// SIMATIC S7-200 project (STEP 7-Micro/WIN), CPU 226 CN REL 02.01

SYMBOL_TABLE INPUT
HMI_ES           I0.0     // HMI急停
WORK_START       I0.1     // 开始工作
BP_ES_RESET      I0.2     // 急停复位
BP_DOOR_RESET    I0.3     // 安全门复位
BP_MANUAL        I0.4     // 手动
BP_AUTO          I0.5     // 自动
BP_START         I0.6     // 启动
ES_OK            I0.7
BP_ES            I1.0     // 操作盒急停
BP_DOOR_PRESET   I1.1     // 安全门预约
AS_OK            I1.2
BP_DOOR_RESET1   I1.3     // 门复位
CS1              I1.4
CS2              I1.5
CS3              I1.6
CS4              I1.7
A伺服就绪            I2.0
A定位结束            I2.1
DSL1             I2.2
DSL2             I2.3
B伺服就绪            I2.4
B定位结束            I2.5
DSR1             I2.6
DSR2             I2.7
BV1_1A           I3.0
BV1_1B           I3.1
BV1_2A           I3.2
BV1_2B           I3.3
BS1              I3.4
BS2              I3.5
B行程保护            I3.6
A请求夹紧            I3.7     // A-R2夹紧请求
BV2_1A           I4.0
BV2_1B           I4.1
BV2_2A           I4.2
BV2_2B           I4.3
BV3_1A           I4.4
BV3_1B           I4.5
BS3              I4.6
B请求夹紧            I4.7     // B-R2夹紧请求
R1_AUTO          I5.0
R1_CYCLE_NO      I5.1
R1_IN_JOB1       I5.2
R1_IN_JOB2       I5.3
R1_HOME          I5.4
R1_ES_OK         I5.5
R1_IN_UNLOAD     I5.6     // 机器人开始抓件
R1_FINISH3       I5.7     // 机器人抓件完成
R1_FINISH1       I6.0     // 机器人放件完成
R1_FINISH2       I6.1     // 机器人取件完成
IN_R1_POS1       I6.2     // 伺服位置返回信号－－产品
IN_R1_POS2       I6.3     // 伺服位置返回信号
IN_R1_POS3       I6.4     // 伺服位置返回信号
IN_R1_POS4       I6.5     // 伺服位置返回信号
IN_R1_PIC1       I6.6     // 机器人返回组信号－－偏差
IN_R1_PIC2       I6.7     // 机器人返回组信号
R2_AUTO          I7.0     // 机器人自动
R2_CYCLE_NO      I7.1     // 机器人上电
R2_IN_JOB1       I7.2
R2_IN_JOB2       I7.3
R2_HOME          I7.4
R2_ES_OK         I7.5     // 机器人急停正常
R2_工位1           I7.6     // A－变位机位置
R2_工位2           I7.7     // B－变位机位置
R2_FINISH1       I8.0     // 机器人2抓件完成
R2_FINISH2       I8.1     // 机器人2焊接完成
IN_R2_POS1       I8.2     // 伺服位置返回信号－－产品
IN_R2_POS2       I8.3     // 伺服位置返回信号
IN_R2_POS3       I8.4     // 伺服位置返回信号
IN_R2_POS4       I8.5     // 伺服位置返回信号
IN_R2_PIC1       I8.6     // 机器人返回组信号－－偏差
IN_R2_PIC2       I8.7     // 机器人返回组信号
AV1_1A           I9.0
AV1_1B           I9.1
AV1_2A           I9.2
AV1_2B           I9.3
AS1              I9.4
AS2              I9.5
A行程保护            I9.6
CV2_A            I9.7     // 横梁传送检测汽缸夹紧信号
AV2_1A           I10.0
AV2_1B           I10.1
AV2_2A           I10.2
AV2_2B           I10.3
AV3_1A           I10.4
AV3_1B           I10.5
AS3              I10.6
END_SYMBOL_TABLE

SYMBOL_TABLE OUTPUT
WORK_H           Q0.0     // 工作指示
ES_H             Q0.1     // 急停复位指示
DOOR_H           Q0.2     // 安全门复位指示
START_H          Q0.3     // 自动启动指示
GN_H             Q0.5     // 绿灯
YE_H             Q0.6     // 黄灯
RD_H             Q0.7     // 红灯
CHECK_DUMMY      Q1.0     // 工件检测虚拟打开
DOOR_OUT         Q1.1     // 安全门
RESET_ES_OUT     Q1.2     // 急停复位输出
RESET_DOOR_OUT   Q1.3
R1_PRO_START     Q4.0     // 给机器人程序开始
RI_CYCLE_START   Q4.1     // 给机器人系统开始
R1_CYCLE_STOP    Q4.2     // 给机器人系统停止
R1_RESET_ES      Q4.3     // 复位机器人急停
R1_JOB1_VAILD    Q4.4     // 开始放件工作的号
R1_JOB2_VAILD    Q4.5     // 开始取件工作的号
R1_STAT1_OK      Q4.6     // 上夹具准备就绪
R1_STAT2_OK      Q4.7     // 下夹具准备就绪
R1_UNLOAD_OK     Q5.0     // 机器人抓件准备就绪
R1_JOB3_VALD     Q5.1     // 启动机器人抓件
R1_POS1          Q5.2     // 伺服位置组信号－－产品
R1_POS2          Q5.3     // 伺服位置组信号
R1_POS3          Q5.4     // 伺服位置组信号
R1_POS4          Q5.5     // 伺服位置组信号
R1_PIC1          Q5.6     // 工件组信号－－偏差
R1_PIC2          Q5.7     // 工件组信号
R2_PRO_START     Q6.0     // 给机器人程序开始
R2_CYCLE_START   Q6.1     // 给机器人系统开始
R2_CYCLE_STOP    Q6.2     // 给机器人系统停止
R2_RESET_ES      Q6.3     // 复位机器人急停
R2_JOB1_VAILD    Q6.4     // 开始放件程序
R2_JOB2_VAILD    Q6.5     // 开始焊接程序
R2_STAT1_OK      Q6.6     // 上夹具准备就绪,可以装件
R2_STAT2_OK      Q6.7     // 下夹具准备就绪,可以装件
R2_A_小件夹紧        Q7.0     // 放小件夹紧A
R2_B_小件夹紧        Q7.1     // 放小件夹紧B
R2_POS1          Q7.2     // 伺服位置组信号－－产品
R2_POS2          Q7.3     // 伺服位置组信号
R2_POS3          Q7.4     // 伺服位置组信号
R2_POS4          Q7.5     // 伺服位置组信号
R2_PIC1          Q7.6     // 工件组信号－－偏差
R2_PIC2          Q7.7     // 工件组信号
AV1_A            Q8.0
AV1_B            Q8.1
AV2_A            Q8.4
AV2_B            Q8.5
AV3_A            Q8.6
AV3_B            Q8.7
BV1_A            Q10.0
BV1_B            Q10.1
BV2_A            Q10.4
BV2_B            Q10.5
BV3_A            Q10.6
BV3_B            Q10.7
A_SRV_ON         Q11.0    // 伺服1使能
A_CLR            Q11.1    // 伺服1报警清除
B_SRV_ON         Q11.2    // 伺服2使能
B_CLR            Q11.3    // 伺服2报警清除
END_SYMBOL_TABLE

SYMBOL_TABLE SERVICE_A
A_MOD_EN         V540.0
A_MAN_RUN        V540.1
A_JOG_P          V540.2
A_JOG_N          V540.3
A_MAN_DIR        V540.4
A_MAN_DONE       V540.5
A_GOTO_START     V540.6
A_GOTO_ABORT     V540.7
A_GOTO_DONE      V541.0
A_RUN_START1     V541.1
A_RUN_ABORT1     V541.2
A_RUN_DONE1      V541.3
A_RUN_START2     V541.4
A_RUN_ABORT2     V541.5
A_RUN_DONE2      V541.6
A_RUN_START3     V541.7
A_RUN_ABORT3     V542.0
A_RUN_DONE3      V542.1
A_RUN_START4     V542.2
A_RUN_ABORT4     V542.3
A_RUN_DONE4      V542.4
A_RUN_START5     V542.5
A_RUN_ABORT5     V542.6
A_RUN_DONE5      V542.7
A_RUN_START6     V543.0
A_RUN_ABORT6     V543.1
A_RUN_DONE6      V543.2
A_RUN_START7     V543.3
A_RUN_ABORT7     V543.4
A_RUN_DONE7      V543.5
A_RUN_START8     V543.6
A_RUN_ABORT8     V543.7
A_RUN_DONE8      V544.0
A_RSEEK_START    V545.0
A_RSEEK_DONE     V545.1
A_DONE           V550.0
A_C_DIR          V550.1
A_ERROR          VB551
A_POS            VD552
A_SPEED          VD556
A_GOTO_ERR       VB560
A_GOTO_C_POS     VD562
A_GOTO_C_SPEED   VD566
A_RUN_ERR        VB570
A_RUN_C_PROF     VB571
A_RUN_C_STEP     VB572
A_RUN_C_POS      VD574
A_RUN_C_SPEED    VD578
A_MAN_SPEED      VD586
A_GOTO_POS       VD590
A_GOTO_SPEED     VD594
A_GOTO_MODE      VB598
A补偿启动            V820.0
A补偿位置            VD822
A补偿速度            VD826
A绝对位置            VD832
A绝对速度            VD836
END_SYMBOL_TABLE

SYMBOL_TABLE UP_A
AV1夹紧的命令         V500.0
AV1夹紧的条件         V500.1
AV1夹紧            V500.2
HMI_AV1夹紧        V500.3
AV1全部夹紧          V500.7
AV1放松的命令         V501.0
AV1放松的条件         V501.1
AV1放松            V501.2
HMI_AV1放松        V501.3
AV1全部放松          V501.7
AV2夹紧的命令         V502.0
AV2夹紧的条件         V502.1
AV2夹紧            V502.2
HMI_AV2夹紧        V502.3
AV2全部夹紧          V502.7
AV2放松的命令         V503.0
AV2放松的条件         V503.1
AV2放松            V503.2
HMI_AV2放松        V503.3
AV2全部放松          V503.7
AV3夹紧的命令         V504.0
AV3夹紧的条件         V504.1
AV3夹紧            V504.2
HMI_AV3夹紧        V504.3
HMI_AV3_MAN_断电   V504.4
AV3全部夹紧          V504.7
AV3放松的命令         V505.0
AV3放松的条件         V505.1
AV3放松            V505.2
HMI_AV3放松        V505.3
AV3全部放松          V505.7
AV大件偏短           V508.0
AV大件偏长           V508.1
AV焊接偏短           V508.2
AV焊接偏长           V508.3
AV取件偏短           V508.4
AV取件偏长           V508.5
AV夹紧             V510.0
AV全部夹紧           V510.1
AV全部放松           V510.2
AV预约             V510.3
AV有小件            V510.4
AV有大件            V510.5
AV有件             V510.6
AV未装件            V510.7
AV放小件准备就绪        V511.0
AV放小件            V511.1
AV请求夹紧           V511.2
AV放小件完成          V511.3
AV放大件准备就绪        V511.4
AV放大件            V511.5
AV放大件完成          V511.6
AV焊接准备就绪         V511.7
AV焊接             V512.0
AV焊接完成           V512.1
AV还原准备           V512.2
AV夹具还原           V512.3
AV取件准备就绪         V512.4
AV取件             V512.5
AV取件完成           V512.6
A_JOB_NUM        VW514
END_SYMBOL_TABLE

SYMBOL_TABLE DOWM_B
BV1夹紧的命令         V600.0
BV1夹紧的条件         V600.1
BV1夹紧            V600.2
HMI_BV1夹紧        V600.3
BV1全部夹紧          V600.7
BV1放松的命令         V601.0
BV1放松的条件         V601.1
BV1放松            V601.2
HMI_BV1放松        V601.3
BV1全部放松          V601.7
BV2夹紧的命令         V602.0
BV2夹紧的条件         V602.1
BV2夹紧            V602.2
HMI_BV2夹紧        V602.3
BV2全部夹紧          V602.7
BV2放松的命令         V603.0
BV2放松的条件         V603.1
BV2放松            V603.2
HMI_BV2放松        V603.3
BV2全部放松          V603.7
BV3夹紧的命令         V604.0
BV3夹紧的条件         V604.1
BV3夹紧            V604.2
HMI_BV3夹紧        V604.3
HMI_BV3_MAN_断电   V604.4
BV3全部夹紧          V604.7
BV3放松的命令         V605.0
BV3放松的条件         V605.1
BV3放松            V605.2
HMI_BV3放松        V605.3
BV3全部放松          V605.7
BV大件偏短           V608.0
BV大件偏长           V608.1
BV焊接偏短           V608.2
BV焊接偏长           V608.3
BV取件偏短           V608.4
BV取件偏长           V608.5
BV夹紧             V610.0
BV全部夹紧           V610.1
BV全部放松           V610.2
BV预约             V610.3
BV有小件            V610.4
BV有大件            V610.5
BV有件             V610.6
BV未装件            V610.7
BV放小件准备就绪        V611.0
BV放小件            V611.1
BV请求夹紧           V611.2
BV放小件完成          V611.3
BV放大件准备就绪        V611.4
BV放大件            V611.5
BV放大件完成          V611.6
BV焊接准备就绪         V611.7
BV焊接             V612.0
BV焊接完成           V612.1
BV还原准备           V612.2
BV夹具还原           V612.3
BV取件准备就绪         V612.4
BV取件             V612.5
BV取件完成           V612.6
B_JOB_NUM        VW614
END_SYMBOL_TABLE

SYMBOL_TABLE SERVICE_B
B_MOD_EN         V640.0
B_MAN_RUN        V640.1
B_JOG_P          V640.2
B_JOG_N          V640.3
B_MAN_DIR        V640.4
B_MAN_DONE       V640.5
B_GOTO_START     V640.6
B_GOTO_ABORT     V640.7
B_GOTO_DONE      V641.0
B_RUN_START1     V641.1
B_RUN_ABORT1     V641.2
B_RUN_DONE1      V641.3
B_RUN_START2     V641.4
B_RUN_ABORT2     V641.5
B_RUN_DONE2      V641.6
B_RUN_START3     V641.7
B_RUN_ABORT3     V642.0
B_RUN_DONE3      V642.1
B_RUN_START4     V642.2
B_RUN_ABORT4     V642.3
B_RUN_DONE4      V642.4
B_RUN_START5     V642.5
B_RUN_ABORT5     V642.6
B_RUN_DONE5      V642.7
B_RUN_START6     V643.0
B_RUN_ABORT6     V643.1
B_RUN_DONE6      V643.2
B_RUN_START7     V643.3
B_RUN_ABORT7     V643.4
B_RUN_DONE7      V643.5
B_RUN_START8     V643.6
B_RUN_ABORT8     V643.7
B_RUN_DONE8      V644.0
B_RSEEK_START    V645.0
B_RSEEK_DONE     V645.1
B_DONE           V650.0
B_C_DIR          V650.1
B_ERROR          VB651
B_POS            VD652
B_SPEED          VD656
B_GOTO_ERR       VB660
B_GOTO_C_POS     VD662
B_GOTO_C_SPEED   VD666
B_RUN_ERR        VB670
B_RUN_C_PROF     VB671
B_RUN_C_STEP     VB672
B_RUN_C_POS      VD674
B_RUN_C_SPEED    VD678
B_MAN_SPEED      VD686
B_GOTO_POS       VD690
B_GOTO_SPEED     VD694
B_GOTO_MODE      VB698
B补偿启动            V920.0
B补偿位置            VD922
B补偿速度            VD926
B绝对位置            VD932
B绝对速度            VD936
END_SYMBOL_TABLE

SYMBOL_TABLE INTERFACE
BV允许抓大件          M4.1
AV允许抓大件          M4.0
开始工作辅助           M0.1
开始工作             M0.0
HMI_RESET_ALARM  M1.0
HMI_LAMP_TEST    M1.1
HMI_RUN_FREE     M1.2
HMI_PAUSE        M1.3
HMI_ST1_PASS     M1.4
HMI_ST2_PASS     M1.5
HMI_INIT         M1.6     // 初始化－HMI
INIT             M1.7
INIT1_FINISH     M2.0
INIT2_FINISH     M2.1
INIT_FINISH      M2.2
PAUSE            M2.3
ST1_PASS         M2.4
ST1_PASS1        M2.5
ST2_PASS         M2.6
ST2_PASS1        M2.7
ST1_WORKING      M3.0
ST2_WORKING      M3.1
HMI_FINISH       M3.2
FINISH           M3.3
PRE_FINISH       M3.4
FINISHED         M3.5
AV_HOME          M3.6
BV_HOME          M3.7
HMI_A_SEV_ON     M5.0
HMI_A_SEV_OFF    M5.1
HMI_A_PIC        M5.2
HMI_B_SEV_ON     M6.0
HMI_B_SEV_OFF    M6.1
HMI_B_PIC        M6.2
绝对画面             M7.0
相对画面             M7.1
HMI_SEV_AB_ON    M8.0
HMI_SEV_AB_HOME  M8.1
NOAUTO           M10.0
AUTO             M10.1
ATUOSTART        M10.2
CONTROL_NO       M10.3
A1合格组信号1         M11.0
A1合格组信号2         M11.1
A2合格组信号1         M11.2
A2合格组信号2         M11.3
B1合格组信号1         M11.4
B1合格组信号2         M11.5
B2合格组信号1         M11.6
B2合格组信号2         M11.7
产品组信号1           M12.0
产品组信号2           M12.1
产品组信号3           M12.2
产品组信号4           M12.3
A工件合格            M14.0
A工件不合格           M14.1
A检测合格            M14.2
B工件合格            M14.4
B工件不合格           M14.5
B检测合格            M14.6
R1_IN_SAFE       M15.0
R1_START         M15.1
R1_JOB_READY     M15.4
R1_POS_OK        M15.5
R1_PIC_OK        M15.6
R1_抓件中           M16.0
R1_抓件完成          M16.1
R2_IN_SAFE       M17.0
R2_START         M17.1
R2_JOB_READY     M17.4
R2_POS_OK        M17.5
R2_PIC_OK        M17.6
A_HOME_POS       M20.0
B_HOME_POS       M22.0
R_IN_SAFE        M23.0
A_CRE_ACT        M30.0
B_CRE_ACT        M30.1
R1_CRE_ACT       M30.2
R2_CRE_ACT       M30.3
SERV_A_ACT       M30.4
SERV_B_ACT       M30.5
DUMMY            M31.0
虚拟               M31.2
虚拟reset          M31.3
PULSE_1          M31.4
HMI_产品选择1        V420.0
HMI_产品选择2        V420.1
HMI_产品选择3        V420.2
HMI_产品选择4        V420.3
HMI_产品选择5        V420.4
HMI_产品选择6        V420.5
HMI_产品选择7        V420.6
HMI_产品选择8        V420.7
HMI_产品选择9        V421.0
HMI_产品选择10       V421.1
HMI_产品选择11       V421.2
HMI_产品选择12       V421.3
HMI_产品选择13       V421.4
HMI_产品选择14       V421.5
HMI_产品选择15       V421.6
HMI_产品选择16       V421.7
产品选择1            V450.0
产品选择2            V450.1
产品选择3            V450.2
产品选择4            V450.3
产品选择5            V450.4
产品选择6            V450.5
产品选择7            V450.6
产品选择8            V450.7
产品选择9            V451.0
产品选择10           V451.1
产品选择11           V451.2
产品选择12           V451.3
产品选择13           V451.4
产品选择14           V451.5
产品选择15           V451.6
产品选择16           V451.7
A产品1             V460.0
A产品2             V460.1
A产品3             V460.2
A产品4             V460.3
A产品5             V460.4
A产品6             V460.5
A产品7             V460.6
A产品8             V460.7
A产品9             V461.0
A产品10            V461.1
A产品11            V461.2
A产品12            V461.3
A产品13            V461.4
A产品14            V461.5
A产品15            V461.6
A产品16            V461.7
B产品1             V462.0
B产品2             V462.1
B产品3             V462.2
B产品4             V462.3
B产品5             V462.4
B产品6             V462.5
B产品7             V462.6
B产品8             V462.7
B产品9             V463.0
B产品10            V463.1
B产品11            V463.2
B产品12            V463.3
B产品13            V463.4
B产品14            V463.5
B产品15            V463.6
B产品16            V463.7
P_放大件            V464.0
P_放小件            V464.1
放大件              V464.2
放小件              V464.3
放件确认             V465.0
放件取消             V465.1
产品选择显示           VB480
产品提示             VB470
选择产品1            V490.0
选择产品2            V490.1
选择产品3            V490.2
选择产品4            V490.3
选择产品5            V490.4
选择产品6            V490.5
选择产品7            V490.6
选择产品8            V490.7
选择产品9            V491.0
选择产品10           V491.1
选择产品11           V491.2
选择产品12           V491.3
选择产品13           V491.4
选择产品14           V491.5
选择产品15           V491.6
选择产品16           V491.7
传送检测气缸信号上        V530.0
检测CS1            V530.1
检测CS2            V530.2
检测CS3            V530.3
END_SYMBOL_TABLE

SYMBOL_TABLE MSSG
AV1_1A_MESS      V400.0
AV1_2A_MESS      V400.1
AV1_3A_MESS      V400.2
AV1_4A_MESS      V400.3
AV1_1B_MESS      V400.4
AV1_2B_MESS      V400.5
AV1_3B_MESS      V400.6
AV1_4B_MESS      V400.7
AV2_1A_MESS      V401.0
AV2_2A_MESS      V401.1
AV2_3A_MESS      V401.2
AV2_4A_MESS      V401.3
AV2_1B_MESS      V401.4
AV2_2B_MESS      V401.5
AV2_3B_MESS      V401.6
AV2_4B_MESS      V401.7
AV3_1A_MESS      V402.0
AV3_2A_MESS      V402.1
AV3_3A_MESS      V402.2
AV3_4A_MESS      V402.3
AV3_1B_MESS      V402.4
AV3_2B_MESS      V402.5
AV3_3B_MESS      V402.6
AV3_4B_MESS      V402.7
AV4_1A_MESS      V403.0
AV4_2A_MESS      V403.1
AV4_3A_MESS      V403.2
AV4_4A_MESS      V403.3
AV4_1B_MESS      V403.4
AV4_2B_MESS      V403.5
AV4_3B_MESS      V403.6
AV4_4B_MESS      V403.7
BV1_1A_MESS      V404.0
BV1_2A_MESS      V404.1
BV1_3A_MESS      V404.2
BV1_4A_MESS      V404.3
BV1_1B_MESS      V404.4
BV1_2B_MESS      V404.5
BV1_3B_MESS      V404.6
BV1_4B_MESS      V404.7
BV2_1A_MESS      V405.0
BV2_2A_MESS      V405.1
BV2_3A_MESS      V405.2
BV2_4A_MESS      V405.3
BV2_1B_MESS      V405.4
BV2_2B_MESS      V405.5
BV2_3B_MESS      V405.6
BV2_4B_MESS      V405.7
BV3_1A_MESS      V406.0
BV3_2A_MESS      V406.1
BV3_3A_MESS      V406.2
BV3_4A_MESS      V406.3
BV3_1B_MESS      V406.4
BV3_2B_MESS      V406.5
BV3_3B_MESS      V406.6
BV3_4B_MESS      V406.7
BV4_1A_MESS      V407.0
BV4_2A_MESS      V407.1
BV4_3A_MESS      V407.2
BV4_4A_MESS      V407.3
BV4_1B_MESS      V407.4
BV4_2B_MESS      V407.5
BV4_3B_MESS      V407.6
BV4_4B_MESS      V407.7
MESS65           V408.0   // 警报   AS1无感应
MESS66           V408.1   // 警报   AS1有感应
MESS67           V408.2   // AS2无感应
MESS68           V408.3   // AS2有感应
MESS69           V408.4   // AS3无感应
MESS70           V408.5   // AS3有感应
MESS71           V408.6   // AS4无感应
MESS72           V408.7   // AS4有感应
MESS73           V409.0   // BS1无感应警报
MESS74           V409.1   // BS1有感应警报
MESS75           V409.2   // BS2无感应
MESS76           V409.3   // BS2有感应
MESS77           V409.4   // BS3无感应
MESS78           V409.5   // BS3有感应
MESS79           V409.6   // BS4无感应
MESS80           V409.7   // BS4有感应
MESS81           V410.0   // CS1无感应警报
MESS82           V410.1   // CS1有感应警报
MESS83           V410.2   // CS2无感应
MESS84           V410.3   // CS2有感应
MESS85           V410.4   // CS3无感应
MESS86           V410.5   // CS3有感应
MESS87           V410.6   // CS4无感应
MESS88           V410.7   // CS4有感应
MESS89           V411.0   // DSL1无感应警报
MESS90           V411.1   // DSL1有感应警报
MESS91           V411.2   // DSL2无感应
MESS92           V411.3   // DSL2有感应
MESS93           V411.4   // DSR1无感应
MESS94           V411.5   // DSR1有感应
MESS95           V411.6   // DSR2无感应
MESS96           V411.7   // DSR2有感应
MESS97           V412.0
MESS98           V412.1
MESS99           V412.2
MESS100          V412.3
MESS101          V412.4
MESS102          V412.5
MESS103          V412.6
MESS104          V412.7
MESS105          V413.0
MESS106          V413.1
MESS107          V413.2
MESS108          V413.3
MESS109          V413.4
MESS110          V413.5
MESS111          V413.6
MESS112          V413.7
MESS113          V414.0   // A伺服电机未查找原点
MESS114          V414.1   // A伺服器未准备就绪
MESS115          V414.2   // A伺服器未上电
MESS116          V414.3   // B伺服电机未查找原点
MESS117          V414.4   // B伺服器未准备就绪
MESS118          V414.5   // B伺服器未上电
MESS119          V414.6   // 机器人1不在原点
MESS120          V414.7   // 机器人2不在原点
MESS121          V415.0   // 机器人1不在自动
MESS122          V415.1   // 机器人2不在自动
MESS123          V415.2   // 机器人1系统未运行
MESS124          V415.3   // 机器人2系统未运行
MESS125          V415.4   // 机器人2不在工位1
MESS126          V415.5   // 机器人2不在工位2
MESS127          V415.6   // A夹具上有工件
MESS128          V415.7   // B夹具上有工件
MESS129          V416.0   // 机器人1急停
MESS130          V416.1   // 机器人2急停
MESS131          V416.2   // 系统急停
MESS132          V416.3   // HMI操作箱急停
MESS133          V416.4   // 安全门操作盒急停
MESS134          V416.5   // 急停按钮未复位
MESS135          V416.6   // 安全打开状态
MESS136          V416.7   // 安全门需要复位
MESS137          V417.0   // 启动条件未满足
MESS138          V417.1
MESS139          V417.2
MESS140          V417.3
MESS141          V417.4
MESS142          V417.5
MESS143          V417.6
MESS144          V417.7
MESS145          V418.0   // 系统空运行测试
MESS146          V418.1   // 夹具1被屏蔽
MESS147          V418.2   // 夹具2被屏蔽
MESS148          V418.3   // 系统暂停运行
MESS149          V418.4   // 系统运行结束
MESS150          V418.5
MESS151          V418.6
MESS152          V418.7
MESS153          V419.0
MESS154          V419.1
MESS155          V419.2
MESS156          V419.3
MESS157          V419.4
MESS158          V419.5
MESS159          V419.6
MESS160          V419.7
AV1_A_CAT        V422.0
AV1_B_CAT        V422.1
AV2_A_CAT        V422.2
AV2_B_CAT        V422.3
AV3_A_CAT        V422.4
AV3_B_CAT        V422.5
AV4_A_CAT        V422.6
AV4_B_CAT        V422.7
BV1_A_CAT        V423.0
BV1_B_CAT        V423.1
BV2_A_CAT        V423.2
BV2_B_CAT        V423.3
BV3_A_CAT        V423.4
BV3_B_CAT        V423.5
BV4_A_CAT        V423.6
BV4_B_CAT        V423.7
AV1_A_RES        V426.0
AV1_B_RES        V426.1
AV2_A_RES        V426.2
AV2_B_RES        V426.3
AV3_A_RES        V426.4
AV3_B_RES        V426.5
AV4_A_RES        V426.6
AV4_B_RES        V426.7
BV1_A_RES        V427.0
BV1_B_RES        V427.1
BV2_A_RES        V427.2
BV2_B_RES        V427.3
BV3_A_RES        V427.4
BV3_B_RES        V427.5
BV4_A_RES        V427.6
BV4_B_RES        V427.7
画面号              VW752
END_SYMBOL_TABLE

ORGANIZATION_BLOCK 主程序:OB1
TITLE=PLC程序用于控制一个自动化生产线，通过两个EM253模块控制松下伺服电机A和B，定位工件长度，并协调搬运机器人和焊接机器人完成生产任务。设备包括松下伺服电机A和B、搬运机器人、焊接机器人、传感器、按钮和指示灯。
// HMI初始化信号由HMI界面触发。系统通过HMI初始化信号启动操作界面，并需确保急停按钮状态未被按下，以保证系统安全运行。操作员可通过手动模式开关或自动模式开关选择运行模式。在手动模式下，操作员可以直接控制夹具的夹紧和放松以及伺服电机的开关。而在自动模式下，启动按钮触发整个生产流程，伺服电机A驱动工位1的工件定位，伺服电机B驱动工位2的工件定位，且需在急停按钮状态正常时激活，以避免设备失控。
// 生产过程中，系统实时监控工位1和工位2的工作状态，并根据A夹具和B夹具的未装件状态判断夹具是否就绪。机器人1开始抓取信号由机器人控制器发出。搬运机器人（机器人1）根据夹具状态执行工件搬运任务，例如，当机器人1开始抓取信号置位时，系统需确认A夹具状态达到指定位置，确保工件正确定位后抓取。随后，焊接机器人（机器人2）在夹具完成夹紧后进行焊接。A夹具工件检测结果用于记录工件长度检测的数据。工件长度检测是关键环节，当传送检测气缸信号为真且工位1和工位2的工作状态均为假时，系统记录A夹具和B夹具的工件检测结果，以确保数据准确。
// 若夹具动作异常，例如伺服电机A的夹紧输出触发失败，A夹具错误计数器会递增以记录异常次数。为了避免误报警影响生产稳定性，系统会在生产周期结束时清零A夹具错误计数器。整个流程结束后，生产周期结束标志置位，系统进入待机状态，等待下一次启动。急停按钮状态若被按下，所有操作立即停止，确保车间人员和设备的安全。
BEGIN
Network 1
LD     SM0.0
CALL   INTERFACE:SBR0
Network 2
LD     SM0.0
CALL   AV1:SBR1
Network 3
LD     SM0.0
CALL   AV2:SBR2
Network 4
LD     SM0.0
CALL   AV3:SBR3
Network 5
LD     SM0.0
CALL   BV1:SBR4
Network 6
LD     SM0.0
CALL   BV2:SBR5
Network 7
LD     SM0.0
CALL   BV3:SBR6
Network 8
LD     A_SRV_ON:Q11.0
CALL   SERVICE_A:SBR7
Network 9
LD     B_SRV_ON:Q11.2
CALL   SERVICEE_B:SBR8
Network 10
LD     SM0.0
CALL   AV:SBR9
Network 11
LD     SM0.0
CALL   BV:SBR10
Network 12
LD     SM0.0
CALL   组信号:SBR22
Network 13
LD     SM0.0
CALL   chanpin:SBR41
Network 14
LD     SM0.0
CALL   PLC_ROBOT1:SBR23
Network 15
LD     SM0.0
CALL   PLC_ROBOT2:SBR24
Network 16
LD     SM0.0
CALL   MESS_2:SBR38
END_ORGANIZATION_BLOCK

SUBROUTINE_BLOCK INTERFACE:SBR0
TITLE=子程序注释
BEGIN
Network 1
LD     SM0.5
EU
LD     SM0.5
ED
OLD
S      PULSE_1:M31.4, 1
Network 2
LD     PULSE_1:M31.4
TON    T200, +2
Network 3
LD     T200
R      PULSE_1:M31.4, 1
Network 4
LD     HMI_INIT:M1.6
EU
A      BP_MANUAL:I0.4
=      INIT:M1.7
Network 5
LD     INIT:M1.7
EU
O      SM0.1
O      ST1_PASS:M2.4
MOVW   +0, VW511
Network 6
LD     INIT:M1.7
EU
O      SM0.1
O      ST2_PASS:M2.6
MOVW   +0, VW611
Network 7
LDW<>  VW511, +0
=      ST1_WORKING:M3.0
Network 8
LDW<>  VW611, +0
=      ST2_WORKING:M3.1
Network 9
LDW=   VW511, +0
A      AV全部放松:V510.2
A      AV未装件:V510.7
=      INIT1_FINISH:M2.0
Network 10
LDW=   VW511, +0
A      AV全部放松:V510.2
=      AV_HOME:M3.6
Network 11
LDW=   VW611, +0
A      BV全部放松:V610.2
A      BV未装件:V610.7
=      INIT2_FINISH:M2.1
Network 12
LDW=   VW611, +0
A      BV全部放松:V610.2
=      BV_HOME:M3.7
Network 13
LD     INIT1_FINISH:M2.0
A      INIT2_FINISH:M2.1
=      INIT_FINISH:M2.2
Network 14
LD     HMI_ST1_PASS:M1.4
EU
A      BP_MANUAL:I0.4
AN     ST1_PASS1:M2.5
LD     HMI_ST1_PASS:M1.4
EU
A      BP_MANUAL:I0.4
A      ST1_PASS1:M2.5
NOT
A      ST1_PASS:M2.4
OLD
=      ST1_PASS:M2.4
Network 15
LD     HMI_ST1_PASS:M1.4
ED
A      BP_MANUAL:I0.4
A      ST1_PASS:M2.4
LD     HMI_ST1_PASS:M1.4
ED
A      BP_MANUAL:I0.4
AN     ST1_PASS:M2.4
NOT
A      ST1_PASS1:M2.5
OLD
=      ST1_PASS1:M2.5
Network 16
LD     HMI_ST2_PASS:M1.5
EU
A      BP_MANUAL:I0.4
AN     ST2_PASS1:M2.7
LD     HMI_ST2_PASS:M1.5
EU
A      BP_MANUAL:I0.4
A      ST2_PASS1:M2.7
NOT
A      ST2_PASS:M2.6
OLD
=      ST2_PASS:M2.6
Network 17
LD     HMI_ST2_PASS:M1.5
ED
A      BP_MANUAL:I0.4
A      ST2_PASS:M2.6
LD     HMI_ST2_PASS:M1.5
ED
A      BP_MANUAL:I0.4
AN     ST2_PASS:M2.6
NOT
A      ST2_PASS1:M2.7
OLD
=      ST2_PASS1:M2.7
Network 18
LD     HMI_PAUSE:M1.3
EU
LD     ST1_WORKING:M3.0
O      ST2_WORKING:M3.1
ALD
A      BP_AUTO:I0.5
LD     WORK_START:I0.1
EU
LD     ST1_WORKING:M3.0
O      ST2_WORKING:M3.1
ALD
A      BP_AUTO:I0.5
LD     INIT_FINISH:M2.2
EU
O      开始工作:M0.0
OLD
NOT
A      PAUSE:M2.3
OLD
=      PAUSE:M2.3
Network 19
LD     HMI_FINISH:M3.2
EU
A      BP_AUTO:I0.5
O      BP_DOOR_PRESET:I1.1
LD     开始工作:M0.0
O      BP_DOOR_RESET:I0.3
NOT
A      PRE_FINISH:M3.4
OLD
=      PRE_FINISH:M3.4
Network 20
LDN    R1_抓件中:M16.0
A      PRE_FINISH:M3.4
LD     开始工作:M0.0
NOT
A      FINISH:M3.3
OLD
=      FINISH:M3.3
Network 21
LD     BV取件完成:V612.6
O      AV取件完成:V512.6
EU
A      R1_HOME:I5.4
A      FINISH:M3.3
S      FINISHED:M3.5, 1
Network 22
LD     FINISHED:M3.5
LD     INIT:M1.7
EU
OLD
LPS
MOVW   +0, VW511
AENO
MOVW   +0, VW512
LPP
MOVW   +0, VW611
AENO
MOVW   +0, VW612
Network 23
LD     开始工作:M0.0
R      FINISHED:M3.5, 1
Network 24
// 网络注释
LD     WORK_START:I0.1
A      BP_AUTO:I0.5
LDN    ST1_PASS:M2.4
AN     ST2_PASS:M2.6
A      INIT_FINISH:M2.2
LDN    ST1_PASS:M2.4
A      ST2_PASS:M2.6
A      INIT1_FINISH:M2.0
OLD
LD     ST1_PASS:M2.4
AN     ST2_PASS:M2.6
A      INIT2_FINISH:M2.1
OLD
ALD
TON    T110, +10
Network 25
LD     WORK_START:I0.1
A      T110
=      开始工作:M0.0
Network 26
LD     ST1_WORKING:M3.0
O      ST2_WORKING:M3.1
LDN    PAUSE:M2.3
LD     PAUSE:M2.3
LD     R1_AUTO:I5.0
AN     R1_CYCLE_NO:I5.1
OLD
LD     R2_AUTO:I7.0
AN     R2_CYCLE_NO:I7.1
OLD
A      SM0.5
OLD
ALD
LDN    ST1_PASS:M2.4
AN     ST2_PASS:M2.6
A      INIT_FINISH:M2.2
LDN    ST1_PASS:M2.4
A      ST2_PASS:M2.6
A      INIT1_FINISH:M2.0
OLD
LD     ST1_PASS:M2.4
AN     ST2_PASS:M2.6
A      INIT2_FINISH:M2.1
OLD
A      PULSE_1:M31.4
OLD
A      BP_AUTO:I0.5
O      HMI_LAMP_TEST:M1.1
=      WORK_H:Q0.0
Network 27
LD     BP_START:I0.6
EU
A      BP_AUTO:I0.5
LD     BP_MANUAL:I0.4
ON     ES_OK:I0.7
ON     AS_OK:I1.2
NOT
A      ATUOSTART:M10.2
OLD
=      ATUOSTART:M10.2
Network 28
LD     ATUOSTART:M10.2
A      R1_AUTO:I5.0
A      R1_CYCLE_NO:I5.1
A      R2_AUTO:I7.0
A      R2_CYCLE_NO:I7.1
LD     R1_AUTO:I5.0
A      R2_AUTO:I7.0
A      BP_AUTO:I0.5
A      SM0.5
OLD
O      HMI_LAMP_TEST:M1.1
=      START_H:Q0.3
Network 29
LDN    ES_OK:I0.7
ON     R1_ES_OK:I5.5
ON     R2_ES_OK:I7.5
A      SM0.5
O      HMI_LAMP_TEST:M1.1
=      ES_H:Q0.1
Network 30
LDN    ES_OK:I0.7
A      BP_ES_RESET:I0.2
=      RESET_ES_OUT:Q1.2
Network 31
LDN    AS_OK:I1.2
A      SM0.5
LD     PRE_FINISH:M3.4
A      PULSE_1:M31.4
OLD
O      HMI_LAMP_TEST:M1.1
=      DOOR_H:Q0.2
Network 32
LDN    AS_OK:I1.2
A      BP_DOOR_RESET:I0.3
=      RESET_DOOR_OUT:Q1.3
Network 33
LD     HMI_A_SEV_ON:M5.0
EU
LD     HMI_SEV_AB_ON:M8.0
EU
OLD
A      BP_MANUAL:I0.4
S      A_SRV_ON:Q11.0, 1
Network 34
LD     HMI_A_SEV_OFF:M5.1
EU
A      BP_MANUAL:I0.4
ON     ES_OK:I0.7
ON     R1_ES_OK:I5.5
ON     R2_ES_OK:I7.5
R      A_SRV_ON:Q11.0, 1
Network 35
LD     HMI_B_SEV_ON:M6.0
EU
LD     HMI_SEV_AB_ON:M8.0
EU
OLD
A      BP_MANUAL:I0.4
S      B_SRV_ON:Q11.2, 1
Network 36
LD     HMI_B_SEV_OFF:M6.1
EU
A      BP_MANUAL:I0.4
ON     ES_OK:I0.7
ON     R1_ES_OK:I5.5
ON     R2_ES_OK:I7.5
R      B_SRV_ON:Q11.2, 1
Network 37
LDN    ES_OK:I0.7
ON     R1_ES_OK:I5.5
ON     R2_ES_OK:I7.5
LD     ES_OK:I0.7
A      R1_ES_OK:I5.5
A      R2_ES_OK:I7.5
AN     AS_OK:I1.2
A      SM0.5
OLD
O      HMI_LAMP_TEST:M1.1
=      RD_H:Q0.7
Network 38
LD     BP_MANUAL:I0.4
LDN    R1_AUTO:I5.0
ON     R2_AUTO:I7.0
A      BP_AUTO:I0.5
O      FINISHED:M3.5
A      SM0.5
OLD
O      HMI_LAMP_TEST:M1.1
=      YE_H:Q0.6
Network 39
LD     ATUOSTART:M10.2
A      R1_AUTO:I5.0
A      R2_AUTO:I7.0
A      R1_CYCLE_NO:I5.1
A      R2_CYCLE_NO:I7.1
LD     ATUOSTART:M10.2
LD     R1_AUTO:I5.0
AN     R1_CYCLE_NO:I5.1
LD     R2_AUTO:I7.0
AN     R2_CYCLE_NO:I7.1
OLD
ALD
A      PULSE_1:M31.4
OLD
LD     FINISH:M3.3
O      FINISHED:M3.5
A      SM0.5
OLD
O      HMI_LAMP_TEST:M1.1
=      GN_H:Q0.5
Network 40
LD     HMI_PAUSE:M1.3
EU
S      PAUSE:M2.3, 1
Network 41
LD     开始工作:M0.0
R      PAUSE:M2.3, 1
Network 43
LD     虚拟:M31.2
A      SM0.5
O      HMI_LAMP_TEST:M1.1
=      CHECK_DUMMY:Q1.0
END_SUBROUTINE_BLOCK

SUBROUTINE_BLOCK AV1:SBR1
TITLE=子程序注释
BEGIN
Network 1 // 网络标题
// 网络注释
LD     SM0.0
A      SM0.0
=      AV1夹紧的命令:V500.0
Network 2
LD     AV2全部夹紧:V502.7
A      AV3全部夹紧:V504.7
A      BP_AUTO:I0.5
=      AV1夹紧的条件:V500.1
Network 3
LD     AV1夹紧的命令:V500.0
A      AV1夹紧的条件:V500.1
EU
A      R2_工位1:I7.6
LD     HMI_AV1夹紧:V500.3
EU
A      BP_MANUAL:I0.4
OLD
=      AV1夹紧:V500.2
Network 4
LD     AV1夹紧:V500.2
LD     AV1放松:V501.2
NOT
A      AV1_A:Q8.0
OLD
=      AV1_A:Q8.0
Network 5
LD     AV1_1A:I9.0
A      AV1_2A:I9.2
=      AV1全部夹紧:V500.7
Network 8
LD     SM0.0
EU
AN     SM0.0
A      SM0.0
A      SM0.0
=      AV1放松的命令:V501.0
Network 9
LD     BP_AUTO:I0.5
=      AV1放松的条件:V501.1
Network 10
LD     AV1放松的命令:V501.0
A      AV1放松的条件:V501.1
LD     AV夹具还原:V512.3
A      AV1放松的条件:V501.1
EU
OLD
A      R2_工位1:I7.6
LD     HMI_AV1放松:V501.3
LD     AV3全部放松:V505.7
A      INIT:M1.7
OLD
EU
A      BP_MANUAL:I0.4
OLD
=      AV1放松:V501.2
Network 11
LD     AV1放松:V501.2
LD     AV1夹紧:V500.2
NOT
A      AV1_B:Q8.1
OLD
=      AV1_B:Q8.1
Network 12
LD     AV1_1B:I9.1
A      AV1_2B:I9.3
=      AV1全部放松:V501.7
END_SUBROUTINE_BLOCK

SUBROUTINE_BLOCK AV2:SBR2
TITLE=子程序注释
BEGIN
Network 1 // 网络标题
// 网络注释
LD     AV请求夹紧:V511.2
=      AV2夹紧的命令:V502.0
Network 2
LD     SM0.0
A      BP_AUTO:I0.5
LD     AV有小件:V510.4
O      HMI_RUN_FREE:M1.2
ALD
=      AV2夹紧的条件:V502.1
Network 3
LD     AV2夹紧的命令:V502.0
A      AV2夹紧的条件:V502.1
EU
LD     HMI_AV2夹紧:V502.3
EU
A      BP_MANUAL:I0.4
OLD
=      AV2夹紧:V502.2
Network 4
LD     AV2夹紧:V502.2
LD     AV2放松:V503.2
NOT
A      AV2_A:Q8.4
OLD
=      AV2_A:Q8.4
Network 5
LD     AV2_1A:I10.0
A      AV2_2A:I10.2
=      AV2全部夹紧:V502.7
Network 8
LD     SM0.0
EU
AN     SM0.0
A      SM0.0
=      AV2放松的命令:V503.0
Network 9
LD     SM0.0
A      BP_AUTO:I0.5
=      AV2放松的条件:V503.1
Network 10
LD     AV2放松的命令:V503.0
A      AV2放松的条件:V503.1
LD     AV夹具还原:V512.3
A      AV2放松的条件:V503.1
EU
OLD
A      R2_工位1:I7.6
LD     HMI_AV2放松:V503.3
O      INIT:M1.7
EU
A      BP_MANUAL:I0.4
OLD
=      AV2放松:V503.2
Network 11
LD     AV2放松:V503.2
LD     AV2夹紧:V502.2
NOT
A      AV2_B:Q8.5
OLD
=      AV2_B:Q8.5
Network 12
LD     AV2_1B:I10.1
A      AV2_2B:I10.3
=      AV2全部放松:V503.7
Network 13 // 网络标题
// 网络注释
END_SUBROUTINE_BLOCK

SUBROUTINE_BLOCK AV3:SBR3
TITLE=子程序注释
BEGIN
Network 1 // 网络标题
// 网络注释
LD     SM0.0
A      AV放大件完成:V511.6
=      AV3夹紧的命令:V504.0
Network 2
LD     AV2全部夹紧:V502.7
A      BP_AUTO:I0.5
LD     AV有大件:V510.5
O      HMI_RUN_FREE:M1.2
ALD
=      AV3夹紧的条件:V504.1
Network 3
LD     AV3夹紧的命令:V504.0
A      AV3夹紧的条件:V504.1
EU
A      R2_工位1:I7.6
LD     HMI_AV3夹紧:V504.3
EU
A      BP_MANUAL:I0.4
OLD
=      AV3夹紧:V504.2
Network 4
LD     AV3夹紧:V504.2
LD     AV3放松:V505.2
LD     HMI_AV3_MAN_断电:V504.4
EU
A      BP_MANUAL:I0.4
OLD
O      AV焊接完成:V512.1
NOT
A      AV3_A:Q8.6
OLD
=      AV3_A:Q8.6
Network 5
LD     AV3_1A:I10.4
=      AV3全部夹紧:V504.7
Network 8
LD     AV取件完成:V512.6
=      AV3放松的命令:V505.0
Network 9
LD     BP_AUTO:I0.5
A      AV1全部放松:V501.7
A      AV2全部放松:V503.7
A      AV未装件:V510.7
=      AV3放松的条件:V505.1
Network 10
LD     AV3放松的命令:V505.0
A      AV3放松的条件:V505.1
EU
LDN    ST2_PASS:M2.6
A      AV夹具还原:V512.3
A      AV3放松的条件:V505.1
EU
OLD
LD     ST2_PASS:M2.6
A      R1_FINISH2:I6.1
A      AV3放松的条件:V505.1
EU
OLD
A      R2_工位1:I7.6
LD     HMI_AV3放松:V505.3
O      INIT:M1.7
EU
A      BP_MANUAL:I0.4
OLD
=      AV3放松:V505.2
Network 11
LD     AV3放松:V505.2
LD     AV3夹紧:V504.2
LD     HMI_AV3_MAN_断电:V504.4
EU
A      BP_MANUAL:I0.4
OLD
NOT
A      AV3_B:Q8.7
OLD
=      AV3_B:Q8.7
Network 12
LD     AV3_1B:I10.5
=      AV3全部放松:V505.7
Network 13 // 网络标题
// 网络注释
END_SUBROUTINE_BLOCK

SUBROUTINE_BLOCK BV1:SBR4
TITLE=子程序注释
BEGIN
Network 1 // 网络标题
// 网络注释
LD     SM0.0
=      BV1夹紧的命令:V600.0
Network 2
LD     BV2全部夹紧:V602.7
A      BV3全部夹紧:V604.7
A      BP_AUTO:I0.5
=      BV1夹紧的条件:V600.1
Network 3
LD     BV1夹紧的命令:V600.0
A      BV1夹紧的条件:V600.1
EU
A      R2_工位2:I7.7
LD     HMI_BV1夹紧:V600.3
EU
A      BP_MANUAL:I0.4
OLD
=      BV1夹紧:V600.2
Network 4
LD     BV1夹紧:V600.2
LD     BV1放松:V601.2
NOT
A      BV1_A:Q10.0
OLD
=      BV1_A:Q10.0
Network 5
LD     BV1_1A:I3.0
A      BV1_2A:I3.2
=      BV1全部夹紧:V600.7
Network 8
LD     SM0.0
EU
AN     SM0.0
A      SM0.0
A      SM0.0
=      BV1放松的命令:V601.0
Network 9
LD     BP_AUTO:I0.5
=      BV1放松的条件:V601.1
Network 10
LD     BV1放松的命令:V601.0
A      BV1放松的条件:V601.1
A      R2_工位2:I7.7
LD     BV夹具还原:V612.3
A      BV1放松的条件:V601.1
A      R2_工位2:I7.7
EU
OLD
LD     HMI_BV1放松:V601.3
LD     BV3全部放松:V605.7
A      INIT:M1.7
OLD
EU
A      BP_MANUAL:I0.4
OLD
=      BV1放松:V601.2
Network 11
LD     BV1放松:V601.2
LD     BV1夹紧:V600.2
NOT
A      BV1_B:Q10.1
OLD
=      BV1_B:Q10.1
Network 12
LD     BV1_1B:I3.1
A      BV1_2B:I3.3
=      BV1全部放松:V601.7
Network 13 // 网络标题
// 网络注释
END_SUBROUTINE_BLOCK

SUBROUTINE_BLOCK BV2:SBR5
TITLE=子程序注释
BEGIN
Network 1 // 网络标题
// 网络注释
LD     BV请求夹紧:V611.2
=      BV2夹紧的命令:V602.0
Network 2
LD     BV有小件:V610.4
O      HMI_RUN_FREE:M1.2
A      BP_AUTO:I0.5
=      BV2夹紧的条件:V602.1
Network 3
LD     BV2夹紧的命令:V602.0
A      BV2夹紧的条件:V602.1
EU
LD     HMI_BV2夹紧:V602.3
EU
A      BP_MANUAL:I0.4
OLD
=      BV2夹紧:V602.2
Network 4
LD     BV2夹紧:V602.2
LD     BV2放松:V603.2
NOT
A      BV2_A:Q10.4
OLD
=      BV2_A:Q10.4
Network 5
LD     BV2_1A:I4.0
A      BV2_2A:I4.2
=      BV2全部夹紧:V602.7
Network 8
LD     SM0.0
EU
AN     SM0.0
A      SM0.0
=      BV2放松的命令:V603.0
Network 9
LD     BP_AUTO:I0.5
=      BV2放松的条件:V603.1
Network 10
LD     BV2放松的命令:V603.0
A      BV2放松的条件:V603.1
EU
A      R2_工位2:I7.7
LD     BV夹具还原:V612.3
A      BV2放松的条件:V603.1
A      R2_工位2:I7.7
EU
OLD
LD     HMI_BV2放松:V603.3
O      INIT:M1.7
EU
A      BP_MANUAL:I0.4
OLD
=      BV2放松:V603.2
Network 11
LD     BV2放松:V603.2
LD     BV2夹紧:V602.2
NOT
A      BV2_B:Q10.5
OLD
=      BV2_B:Q10.5
Network 12
LD     BV2_1B:I4.1
A      BV2_2B:I4.3
=      BV2全部放松:V603.7
Network 13 // 网络标题
// 网络注释
END_SUBROUTINE_BLOCK

SUBROUTINE_BLOCK BV3:SBR6
TITLE=子程序注释
BEGIN
Network 1 // 网络标题
// 网络注释
LD     BV放大件完成:V611.6
=      BV3夹紧的命令:V604.0
Network 2
LD     BV2全部夹紧:V602.7
A      BP_AUTO:I0.5
LD     BV有大件:V610.5
O      HMI_RUN_FREE:M1.2
ALD
=      BV3夹紧的条件:V604.1
Network 3
LD     BV3夹紧的命令:V604.0
A      BV3夹紧的条件:V604.1
EU
A      R2_工位2:I7.7
LD     HMI_BV3夹紧:V604.3
EU
A      BP_MANUAL:I0.4
OLD
=      BV3夹紧:V604.2
Network 4
LD     BV3夹紧:V604.2
LD     BV3放松:V605.2
LD     BP_MANUAL:I0.4
A      HMI_BV3_MAN_断电:V604.4
EU
OLD
O      BV焊接完成:V612.1
NOT
A      BV3_A:Q10.6
OLD
=      BV3_A:Q10.6
Network 5
LD     BV3_1A:I4.4
=      BV3全部夹紧:V604.7
Network 8
LD     BV取件完成:V612.6
=      BV3放松的命令:V605.0
Network 9
LD     BV1全部放松:V601.7
A      BV2全部放松:V603.7
A      BV未装件:V610.7
A      BP_AUTO:I0.5
=      BV3放松的条件:V605.1
Network 10
LD     BV3放松的命令:V605.0
A      BV3放松的条件:V605.1
EU
LDN    ST1_PASS:M2.4
A      BV夹具还原:V612.3
A      BV3放松的条件:V605.1
EU
OLD
LD     ST1_PASS:M2.4
A      R1_FINISH2:I6.1
A      BV3放松的条件:V605.1
EU
OLD
A      R2_工位2:I7.7
LD     HMI_BV3放松:V605.3
O      INIT:M1.7
EU
A      BP_MANUAL:I0.4
OLD
=      BV3放松:V605.2
Network 11
LD     BV3放松:V605.2
LD     BV3夹紧:V604.2
LD     HMI_BV3_MAN_断电:V604.4
A      BP_MANUAL:I0.4
EU
OLD
NOT
A      BV3_B:Q10.7
OLD
=      BV3_B:Q10.7
Network 12
LD     BV3_1B:I4.5
=      BV3全部放松:V605.7
Network 13 // 网络标题
// 网络注释
END_SUBROUTINE_BLOCK

SUBROUTINE_BLOCK SERVICE_A:SBR7
TITLE=子程序注释
BEGIN
Network 1
LD     SM0.0
=      L60.0
LD     SM0.0
=      L63.7
LD     L60.0
CALL   POS0_CTRL:SBR11, L63.7, A_DONE:V550.0, A_ERROR:VB551, A_POS:VD552, A_SPEED:VD556, A_C_DIR:V550.1
Network 2
LDR>=  A_MAN_SPEED:VD586, 30.0
MOVR   30.0, A_MAN_SPEED:VD586
Network 3
LD     SM0.0
A      BP_MANUAL:I0.4
A      AV未装件:V510.7
A      A_SRV_ON:Q11.0
A      A_RSEEK_DONE:V545.1
=      L60.0
LD     A_MAN_RUN:V540.1
AN     A_JOG_P:V540.2
AN     A_JOG_N:V540.3
=      L63.7
LD     A_JOG_P:V540.2
AN     A_MAN_RUN:V540.1
AN     A_JOG_N:V540.3
=      L63.6
LD     A_JOG_N:V540.3
AN     A_MAN_RUN:V540.1
AN     A_JOG_P:V540.2
=      L63.5
LD     L60.0
CALL   POS0_MAN:SBR12, L63.7, L63.6, L63.5, A_MAN_SPEED:VD586, A_MAN_DIR:V540.4, A_ERROR:VB551, A_POS:VD552, A_SPEED:VD556, A_C_DIR:V550.1
Network 4
LDD=   A_POS:VD552, +0
A      A_RSEEK_DONE:V545.1
=      A_HOME_POS:M20.0
Network 5
LDW=   画面号:VW752, +14
OW=    画面号:VW752, +15
=      绝对画面:M7.0
Network 6
LD     绝对画面:M7.0
MOVB   0, A_GOTO_MODE:VB598
Network 7
LDW=   画面号:VW752, +12
=      相对画面:M7.1
Network 8
LD     相对画面:M7.1
MOVB   1, A_GOTO_MODE:VB598
Network 9
LD     绝对画面:M7.0
MOVD   A绝对位置:VD832, A_GOTO_POS:VD590
MOVD   A绝对速度:VD836, A_GOTO_SPEED:VD594
Network 10
LDR>=  A补偿速度:VD826, 1.0
MOVR   1.0, A补偿速度:VD826
Network 11
LDR<=  A补偿位置:VD822, -3.0
AR>=   A补偿位置:VD822, 3.0
MOVR   1.0, A补偿位置:VD822
Network 12
LD     相对画面:M7.1
MOVD   A补偿位置:VD822, A_GOTO_POS:VD590
MOVD   A补偿速度:VD826, A_GOTO_SPEED:VD594
Network 13
LDR>=  A_GOTO_SPEED:VD594, 30.0
MOVR   30.0, A_GOTO_SPEED:VD594
Network 14
LD     SM0.0
A      BP_MANUAL:I0.4
A      A_SRV_ON:Q11.0
A      A_RSEEK_DONE:V545.1
=      L60.0
LD     A_GOTO_START:V540.6
EU
A      绝对画面:M7.0
LD     A补偿启动:V820.0
EU
A      相对画面:M7.1
OLD
=      L63.7
LD     L60.0
CALL   POS0_GOTO:SBR13, L63.7, A_GOTO_POS:VD590, A_GOTO_SPEED:VD594, A_GOTO_MODE:VB598, A_GOTO_ABORT:V540.7, A_GOTO_DONE:V541.0, A_GOTO_ERR:VB560, A_GOTO_C_POS:VD562, A_GOTO_C_SPEED:VD566
Network 15
LD     SM0.0
A      BP_MANUAL:I0.4
A      AV未装件:V510.7
A      A_SRV_ON:Q11.0
A      R1_IN_SAFE:M15.0
A      R2_IN_SAFE:M17.0
=      L60.0
LD     A_RSEEK_START:V545.0
EU
=      L63.7
LD     L60.0
CALL   POS0_RSEEK:SBR15, L63.7, A_RSEEK_DONE:V545.1, A_ERROR:VB551
Network 16
LD     SM0.0
A      A_SRV_ON:Q11.0
A      A_RSEEK_DONE:V545.1
AN     AS2:I9.5
LD     选择产品1:V490.0
O      选择产品2:V490.1
ALD
=      L60.0
LD     产品选择1:V450.0
EU
LD     产品选择2:V450.1
EU
OLD
A      BP_MANUAL:I0.4
=      L63.7
LD     L60.0
CALL   POS0_RUN:SBR14, L63.7, Profile0_2340:VB364, A_RUN_ABORT1:V541.2, A_RUN_DONE1:V541.3, A_RUN_ERR:VB570, A_RUN_C_PROF:VB571, A_RUN_C_STEP:VB572, A_RUN_C_POS:VD574, A_RUN_C_SPEED:VD578
Network 17
LD     SM0.0
A      A_SRV_ON:Q11.0
A      A_RSEEK_DONE:V545.1
AN     AS2:I9.5
LD     选择产品3:V490.2
O      选择产品4:V490.3
ALD
=      L60.0
LD     产品选择3:V450.2
EU
LD     产品选择4:V450.3
EU
OLD
A      BP_MANUAL:I0.4
=      L63.7
LD     L60.0
CALL   POS0_RUN:SBR14, L63.7, Profile0_2390:VB365, A_RUN_ABORT2:V541.5, A_RUN_DONE2:V541.6, A_RUN_ERR:VB570, A_RUN_C_PROF:VB571, A_RUN_C_STEP:VB572, A_RUN_C_POS:VD574, A_RUN_C_SPEED:VD578
Network 18
LD     SM0.0
A      A_SRV_ON:Q11.0
A      A_RSEEK_DONE:V545.1
AN     AS2:I9.5
LD     选择产品5:V490.4
O      选择产品6:V490.5
ALD
=      L60.0
LD     产品选择5:V450.4
EU
LD     产品选择6:V450.5
EU
OLD
A      BP_MANUAL:I0.4
=      L63.7
LD     L60.0
CALL   POS0_RUN:SBR14, L63.7, Profile0_2440:VB366, A_RUN_ABORT3:V542.0, A_RUN_DONE3:V542.1, A_RUN_ERR:VB570, A_RUN_C_PROF:VB571, A_RUN_C_STEP:VB572, A_RUN_C_POS:VD574, A_RUN_C_SPEED:VD578
Network 19
LD     SM0.0
A      A_SRV_ON:Q11.0
A      A_RSEEK_DONE:V545.1
AN     AS2:I9.5
LD     选择产品7:V490.6
O      选择产品8:V490.7
ALD
=      L60.0
LD     产品选择7:V450.6
EU
LD     产品选择8:V450.7
EU
OLD
A      BP_MANUAL:I0.4
=      L63.7
LD     L60.0
CALL   POS0_RUN:SBR14, L63.7, Profile0_2790:VB367, A_RUN_ABORT4:V542.3, A_RUN_DONE4:V542.4, A_RUN_ERR:VB570, A_RUN_C_PROF:VB571, A_RUN_C_STEP:VB572, A_RUN_C_POS:VD574, A_RUN_C_SPEED:VD578
Network 20
LD     SM0.0
A      A_SRV_ON:Q11.0
A      A_RSEEK_DONE:V545.1
AN     AS2:I9.5
LD     选择产品9:V491.0
O      选择产品10:V491.1
ALD
=      L60.0
LD     产品选择9:V451.0
EU
LD     产品选择10:V451.1
EU
OLD
A      BP_MANUAL:I0.4
=      L63.7
LD     L60.0
CALL   POS0_RUN:SBR14, L63.7, Profile0_2370:VB368, A_RUN_ABORT5:V542.6, A_RUN_DONE5:V542.7, A_RUN_ERR:VB570, A_RUN_C_PROF:VB571, A_RUN_C_STEP:VB572, A_RUN_C_POS:VD574, A_RUN_C_SPEED:VD578
Network 21
LD     SM0.0
A      A_SRV_ON:Q11.0
A      A_RSEEK_DONE:V545.1
AN     AS2:I9.5
A      选择产品11:V491.2
=      L60.0
LD     产品选择11:V451.2
EU
A      BP_MANUAL:I0.4
=      L63.7
LD     L60.0
CALL   POS0_RUN:SBR14, L63.7, Profile0_2420:VB369, A_RUN_ABORT6:V543.1, A_RUN_DONE6:V543.2, A_RUN_ERR:VB570, A_RUN_C_PROF:VB571, A_RUN_C_STEP:VB572, A_RUN_C_POS:VD574, A_RUN_C_SPEED:VD578
Network 22
LD     SM0.0
A      A_SRV_ON:Q11.0
A      A_RSEEK_DONE:V545.1
AN     AS2:I9.5
A      选择产品12:V491.3
=      L60.0
LD     产品选择12:V451.3
EU
A      BP_MANUAL:I0.4
=      L63.7
LD     L60.0
CALL   POS0_RUN:SBR14, L63.7, Profile0_2470:VB370, A_RUN_ABORT7:V543.4, A_RUN_DONE7:V543.5, A_RUN_ERR:VB570, A_RUN_C_PROF:VB571, A_RUN_C_STEP:VB572, A_RUN_C_POS:VD574, A_RUN_C_SPEED:VD578
Network 23
LD     SM0.0
A      A_SRV_ON:Q11.0
A      A_RSEEK_DONE:V545.1
AN     AS2:I9.5
LD     选择产品13:V491.4
O      选择产品14:V491.5
ALD
=      L60.0
LD     产品选择13:V451.4
EU
LD     产品选择14:V451.5
EU
OLD
A      BP_MANUAL:I0.4
=      L63.7
LD     L60.0
CALL   POS0_RUN:SBR14, L63.7, Profile0_2820:VB371, A_RUN_ABORT8:V543.7, A_RUN_DONE8:V544.0, A_RUN_ERR:VB570, A_RUN_C_PROF:VB571, A_RUN_C_STEP:VB572, A_RUN_C_POS:VD574, A_RUN_C_SPEED:VD578
END_SUBROUTINE_BLOCK

SUBROUTINE_BLOCK SERVICEE_B:SBR8
TITLE=子程序注释
BEGIN
Network 1 // 网络标题
// 网络注释
LD     SM0.0
=      L60.0
LD     SM0.0
=      L63.7
LD     L60.0
CALL   POS1_CTRL:SBR26, L63.7, B_DONE:V650.0, B_ERROR:VB651, B_POS:VD652, B_SPEED:VD656, B_C_DIR:V650.1
Network 2
LDD=   B_POS:VD652, +0
A      B_RSEEK_DONE:V645.1
=      B_HOME_POS:M22.0
Network 3
LDR>=  B_MAN_SPEED:VD686, 30.0
MOVR   30.0, B_MAN_SPEED:VD686
Network 4
LD     SM0.0
A      BP_MANUAL:I0.4
A      BV未装件:V610.7
A      B_SRV_ON:Q11.2
A      B_RSEEK_DONE:V645.1
=      L60.0
LD     B_MAN_RUN:V640.1
AN     B_JOG_P:V640.2
AN     B_JOG_N:V640.3
=      L63.7
LD     B_JOG_P:V640.2
AN     B_MAN_RUN:V640.1
AN     B_JOG_N:V640.3
=      L63.6
LD     B_JOG_N:V640.3
AN     B_MAN_RUN:V640.1
AN     B_JOG_P:V640.2
=      L63.5
LD     L60.0
CALL   POS1_MAN:SBR27, L63.7, L63.6, L63.5, B_MAN_SPEED:VD686, B_MAN_DIR:V640.4, B_ERROR:VB651, B_POS:VD652, B_SPEED:VD656, B_C_DIR:V650.1
Network 5
LD     相对画面:M7.1
MOVB   1, B_GOTO_MODE:VB698
Network 6
LD     绝对画面:M7.0
MOVD   B绝对位置:VD932, B_GOTO_POS:VD690
MOVD   B绝对速度:VD936, B_GOTO_SPEED:VD694
Network 7
LDR>=  B补偿速度:VD926, 1.0
MOVR   1.0, B补偿速度:VD926
Network 8
LDR<=  B补偿位置:VD922, -3.0
AR>=   B补偿位置:VD922, 3.0
MOVR   3.0, B补偿位置:VD922
Network 9
LD     相对画面:M7.1
MOVD   B补偿位置:VD922, B_GOTO_POS:VD690
MOVD   B补偿速度:VD926, B_GOTO_SPEED:VD694
Network 10
LDR>=  B_GOTO_SPEED:VD694, 30.0
MOVR   30.0, B_GOTO_SPEED:VD694
Network 11
LD     SM0.0
A      BP_MANUAL:I0.4
A      B_SRV_ON:Q11.2
A      B_RSEEK_DONE:V645.1
=      L60.0
LD     B_GOTO_START:V640.6
EU
A      绝对画面:M7.0
LD     B补偿启动:V920.0
EU
A      相对画面:M7.1
OLD
=      L63.7
LD     L60.0
CALL   POS1_GOTO:SBR28, L63.7, B_GOTO_POS:VD690, B_GOTO_SPEED:VD694, B_GOTO_MODE:VB698, B_GOTO_ABORT:V640.7, B_GOTO_DONE:V641.0, B_GOTO_ERR:VB660, B_GOTO_C_POS:VD662, B_GOTO_C_SPEED:VD666
Network 12
LD     SM0.0
A      BP_MANUAL:I0.4
A      BV未装件:V610.7
A      B_SRV_ON:Q11.2
A      R1_IN_SAFE:M15.0
A      R2_IN_SAFE:M17.0
=      L60.0
LD     B_RSEEK_START:V645.0
EU
=      L63.7
LD     L60.0
CALL   POS1_RSEEK:SBR30, L63.7, B_RSEEK_DONE:V645.1, B_ERROR:VB651
Network 13
LD     SM0.0
A      B_SRV_ON:Q11.2
A      B_RSEEK_DONE:V645.1
AN     BS2:I3.5
LD     选择产品1:V490.0
O      选择产品2:V490.1
ALD
=      L60.0
LD     产品选择1:V450.0
EU
LD     产品选择2:V450.1
EU
OLD
A      BP_MANUAL:I0.4
=      L63.7
LD     L60.0
CALL   POS1_RUN:SBR29, L63.7, Profile1_2340:VB1677, B_RUN_ABORT1:V641.2, B_RUN_DONE1:V641.3, B_RUN_ERR:VB670, B_RUN_C_PROF:VB671, B_RUN_C_STEP:VB672, B_RUN_C_POS:VD674, B_RUN_C_SPEED:VD678
Network 14
LD     SM0.0
A      B_SRV_ON:Q11.2
A      B_RSEEK_DONE:V645.1
AN     BS2:I3.5
LD     选择产品3:V490.2
O      选择产品4:V490.3
ALD
=      L60.0
LD     产品选择3:V450.2
EU
LD     产品选择4:V450.3
EU
OLD
A      BP_MANUAL:I0.4
=      L63.7
LD     L60.0
CALL   POS1_RUN:SBR29, L63.7, Profile1_2390:VB1678, B_RUN_ABORT2:V641.5, B_RUN_DONE2:V641.6, B_RUN_ERR:VB670, B_RUN_C_PROF:VB671, B_RUN_C_STEP:VB672, B_RUN_C_POS:VD674, B_RUN_C_SPEED:VD678
Network 15
LD     SM0.0
A      B_SRV_ON:Q11.2
A      B_RSEEK_DONE:V645.1
AN     BS2:I3.5
LD     选择产品5:V490.4
O      选择产品6:V490.5
ALD
=      L60.0
LD     产品选择5:V450.4
EU
LD     产品选择6:V450.5
EU
OLD
A      BP_MANUAL:I0.4
=      L63.7
LD     L60.0
CALL   POS1_RUN:SBR29, L63.7, Profile1_2440:VB1679, B_RUN_ABORT3:V642.0, B_RUN_DONE3:V642.1, B_RUN_ERR:VB670, B_RUN_C_PROF:VB671, B_RUN_C_STEP:VB672, B_RUN_C_POS:VD674, B_RUN_C_SPEED:VD678
Network 16
LD     SM0.0
A      B_SRV_ON:Q11.2
A      B_RSEEK_DONE:V645.1
AN     BS2:I3.5
LD     选择产品7:V490.6
O      选择产品8:V490.7
ALD
=      L60.0
LD     产品选择7:V450.6
EU
LD     产品选择8:V450.7
EU
OLD
A      BP_MANUAL:I0.4
=      L63.7
LD     L60.0
CALL   POS1_RUN:SBR29, L63.7, Profile1_2790:VB1680, B_RUN_ABORT4:V642.3, B_RUN_DONE4:V642.4, B_RUN_ERR:VB670, B_RUN_C_PROF:VB671, B_RUN_C_STEP:VB672, B_RUN_C_POS:VD674, B_RUN_C_SPEED:VD678
Network 17
LD     SM0.0
A      B_SRV_ON:Q11.2
A      B_RSEEK_DONE:V645.1
AN     BS2:I3.5
LD     选择产品9:V491.0
O      选择产品10:V491.1
ALD
=      L60.0
LD     产品选择9:V451.0
EU
LD     产品选择10:V451.1
EU
OLD
A      BP_MANUAL:I0.4
=      L63.7
LD     L60.0
CALL   POS1_RUN:SBR29, L63.7, Profile1_2370:VB1681, B_RUN_ABORT5:V642.6, B_RUN_DONE5:V642.7, B_RUN_ERR:VB670, B_RUN_C_PROF:VB671, B_RUN_C_STEP:VB672, B_RUN_C_POS:VD674, B_RUN_C_SPEED:VD678
Network 18
LD     SM0.0
A      B_SRV_ON:Q11.2
A      B_RSEEK_DONE:V645.1
AN     BS2:I3.5
A      选择产品11:V491.2
=      L60.0
LD     产品选择11:V451.2
EU
A      BP_MANUAL:I0.4
=      L63.7
LD     L60.0
CALL   POS1_RUN:SBR29, L63.7, Profile1_2420:VB1682, B_RUN_ABORT6:V643.1, B_RUN_DONE6:V643.2, B_RUN_ERR:VB670, B_RUN_C_PROF:VB671, B_RUN_C_STEP:VB672, B_RUN_C_POS:VD674, B_RUN_C_SPEED:VD678
Network 19
LD     SM0.0
A      B_SRV_ON:Q11.2
A      B_RSEEK_DONE:V645.1
AN     BS2:I3.5
A      选择产品12:V491.3
=      L60.0
LD     产品选择12:V451.3
EU
A      BP_MANUAL:I0.4
=      L63.7
LD     L60.0
CALL   POS1_RUN:SBR29, L63.7, Profile1_2470:VB1683, B_RUN_ABORT7:V643.4, B_RUN_DONE7:V643.5, B_RUN_ERR:VB670, B_RUN_C_PROF:VB671, B_RUN_C_STEP:VB672, B_RUN_C_POS:VD674, B_RUN_C_SPEED:VD678
Network 20
LD     SM0.0
A      B_SRV_ON:Q11.2
A      B_RSEEK_DONE:V645.1
AN     BS2:I3.5
LD     选择产品13:V491.4
O      选择产品14:V491.5
ALD
=      L60.0
LD     产品选择13:V451.4
EU
LD     产品选择14:V451.5
EU
OLD
A      BP_MANUAL:I0.4
=      L63.7
LD     L60.0
CALL   POS1_RUN:SBR29, L63.7, Profile1_2820:VB1684, B_RUN_ABORT8:V643.7, B_RUN_DONE8:V644.0, B_RUN_ERR:VB670, B_RUN_C_PROF:VB671, B_RUN_C_STEP:VB672, B_RUN_C_POS:VD674, B_RUN_C_SPEED:VD678
END_SUBROUTINE_BLOCK

SUBROUTINE_BLOCK AV:SBR9
TITLE=子程序注释
BEGIN
Network 1 // 网络标题
// 网络注释
LD     AV1全部夹紧:V500.7
A      AV2全部夹紧:V502.7
A      AV3全部夹紧:V504.7
=      AV全部夹紧:V510.1
Network 2
LD     AV1全部放松:V501.7
A      AV2全部放松:V503.7
A      AV3全部放松:V505.7
=      AV全部放松:V510.2
Network 3
LD     AS1:I9.4
A      AS3:I10.6
=      AV有小件:V510.4
Network 4
LD     AS2:I9.5
=      AV有大件:V510.5
Network 5
LD     AV有小件:V510.4
A      AV有大件:V510.5
=      AV有件:V510.6
Network 6
LDN    AS1:I9.4
AN     AS2:I9.5
AN     AS3:I10.6
=      AV未装件:V510.7
Network 7
LDW=   A_JOB_NUM:VW514, +2
OW=    A_JOB_NUM:VW514, +3
=      A工件合格:M14.0
Network 8
LDW=   VW520, +1
OW=    VW520, +4
=      A工件不合格:M14.1
Network 9
LDW=   VW520, +2
OW=    VW520, +3
=      A检测合格:M14.2
Network 10
LDW=   A_JOB_NUM:VW514, +2
=      AV大件偏短:V508.0
Network 11
LDW=   A_JOB_NUM:VW514, +3
=      AV大件偏长:V508.1
Network 12
LDW=   VW516, +2
=      AV焊接偏短:V508.2
Network 13
LDW=   VW516, +3
=      AV焊接偏长:V508.3
Network 14
LDW=   VW518, +2
=      AV取件偏短:V508.4
Network 15
LDW=   VW518, +3
=      AV取件偏长:V508.5
Network 16
LD     A工件不合格:M14.1
A      BP_AUTO:I0.5
R      A1合格组信号1:M11.0, 2
S      A1合格组信号1:M11.0, 1
Network 17
LD     AV大件偏短:V508.0
O      AV取件偏短:V508.4
A      BP_AUTO:I0.5
R      A1合格组信号1:M11.0, 2
S      A1合格组信号2:M11.1, 1
Network 18
LD     AV大件偏长:V508.1
O      AV取件偏长:V508.5
O      A检测合格:M14.2
A      BP_AUTO:I0.5
S      A1合格组信号1:M11.0, 2
Network 19
LD     BP_MANUAL:I0.4
O      AV放大件完成:V511.6
O      AV取件完成:V512.6
ON     CS4:I1.7
R      A1合格组信号1:M11.0, 2
Network 20
LD     AV焊接偏短:V508.2
A      BP_AUTO:I0.5
R      A2合格组信号1:M11.2, 2
S      A2合格组信号2:M11.3, 1
Network 21
LD     AV焊接偏长:V508.3
A      BP_AUTO:I0.5
S      A2合格组信号1:M11.2, 2
Network 22
LD     BP_MANUAL:I0.4
O      AV焊接完成:V512.1
R      A2合格组信号1:M11.2, 2
Network 23
LD     AV全部放松:V510.2
EU
A      AV取件完成:V512.6
AN     ST1_PASS:M2.4
MOVW   +0, VW512
MOVW   +0, VW511
Network 24
// 网络注释
LD     AV全部放松:V510.2
A      AV未装件:V510.7
A      BP_AUTO:I0.5
LD     开始工作:M0.0
AN     ST1_PASS:M2.4
LDN    FINISH:M3.3
A      BV焊接完成:V612.1
AN     ST2_PASS:M2.6
OLD
LDN    FINISH:M3.3
A      R1_HOME:I5.4
A      ST2_PASS:M2.6
OLD
ALD
LDN    HMI_RUN_FREE:M1.2
A      DSL1:I2.2
A      DSR1:I2.6
LD     HMI_RUN_FREE:M1.2
AN     DSL1:I2.2
AN     DSR1:I2.6
OLD
ALD
AW=    VW511, +0
EU
AN     R2_IN_JOB1:I7.2
AN     AV放小件准备就绪:V511.0
A      R2_工位1:I7.6
LD     BP_MANUAL:I0.4
ON     AV全部放松:V510.2
ON     AV未装件:V510.7
LDN    HMI_RUN_FREE:M1.2
LDN    DSL1:I2.2
ON     DSR1:I2.6
ALD
OLD
LD     HMI_RUN_FREE:M1.2
LD     DSL1:I2.2
O      DSR1:I2.6
ALD
OLD
LD     AV放小件:V511.1
EU
OLD
NOT
A      AV放小件准备就绪:V511.0
OLD
=      AV放小件准备就绪:V511.0
Network 25
LD     R2_IN_JOB1:I7.2
EU
A      AV放小件准备就绪:V511.0
A      R2_AUTO:I7.0
LDW<>  VW611, +0
AN     ST2_PASS:M2.6
A      BV还原准备:V612.2
OW=    VW611, +0
O      ST2_PASS:M2.6
A      AV放小件完成:V511.3
EU
NOT
A      AV放小件:V511.1
OLD
=      AV放小件:V511.1
Network 26
LD     A请求夹紧:I3.7
EU
A      AV放小件:V511.1
A      R2_AUTO:I7.0
LD     AV放小件完成:V511.3
EU
NOT
A      AV请求夹紧:V511.2
OLD
=      AV请求夹紧:V511.2
Network 27
LD     R2_FINISH1:I8.0
EU
A      AV放小件:V511.1
A      R2_AUTO:I7.0
LD     AV放大件:V511.5
EU
NOT
A      AV放小件完成:V511.3
OLD
=      AV放小件完成:V511.3
Network 28
LD     AV放小件完成:V511.3
A      AV1全部放松:V501.7
A      AV2全部夹紧:V502.7
A      AV3全部放松:V505.7
LD     AV有小件:V510.4
O      HMI_RUN_FREE:M1.2
ALD
AN     AV有大件:V510.5
A      R1_抓件完成:M16.1
A      BP_AUTO:I0.5
A      R2_工位1:I7.6
EU
LD     BP_MANUAL:I0.4
ON     AV1全部放松:V501.7
ON     AV2全部夹紧:V502.7
ON     AV3全部放松:V505.7
LDN    HMI_RUN_FREE:M1.2
LDN    AV有小件:V510.4
O      AS2:I9.5
ALD
OLD
LD     AV放大件:V511.5
EU
OLD
NOT
A      AV放大件准备就绪:V511.4
OLD
=      AV放大件准备就绪:V511.4
Network 29
LD     R1_IN_JOB1:I5.2
EU
A      AV放大件准备就绪:V511.4
A      R1_AUTO:I5.0
LD     AV放大件完成:V511.6
EU
NOT
A      AV放大件:V511.5
OLD
=      AV放大件:V511.5
Network 30
LD     AV放大件:V511.5
EU
A      R2_AUTO:I7.0
AW<>   VW611, +0
AN     ST2_PASS:M2.6
LD     BV夹具还原:V612.3
EU
NOT
A      BV还原准备:V612.2
OLD
=      BV还原准备:V612.2
Network 31
LD     R1_FINISH1:I6.0
EU
A      AV放大件:V511.5
A      R1_AUTO:I5.0
LD     AV全部夹紧:V510.1
LD     AV有件:V510.6
O      HMI_RUN_FREE:M1.2
ALD
EU
NOT
A      AV放大件完成:V511.6
OLD
=      AV放大件完成:V511.6
Network 32
LD     AV全部夹紧:V510.1
LD     AV有件:V510.6
O      HMI_RUN_FREE:M1.2
ALD
EU
A      BP_AUTO:I0.5
A      R2_工位1:I7.6
A      R2_IN_SAFE:M17.0
LDN    AV全部夹紧:V510.1
LDN    HMI_RUN_FREE:M1.2
AN     AV有件:V510.6
OLD
LD     AV焊接:V512.0
EU
OLD
NOT
A      AV焊接准备就绪:V511.7
OLD
=      AV焊接准备就绪:V511.7
Network 33
LD     R2_IN_JOB2:I7.3
EU
A      AV焊接准备就绪:V511.7
A      R2_AUTO:I7.0
LD     AV焊接完成:V512.1
EU
NOT
A      AV焊接:V512.0
OLD
=      AV焊接:V512.0
Network 34
LD     R2_FINISH2:I8.1
EU
A      AV焊接:V512.0
A      R2_AUTO:I7.0
LD     AV夹具还原:V512.3
EU
NOT
A      AV焊接完成:V512.1
OLD
=      AV焊接完成:V512.1
Network 35
LDN    ST2_PASS:M2.6
A      R2_工位1:I7.6
A      AV还原准备:V512.2
O      ST2_PASS:M2.6
LDN    ST2_PASS:M2.6
A      R2_工位1:I7.6
A      FINISH:M3.3
OLD
A      AV焊接完成:V512.1
EU
A      BP_AUTO:I0.5
LD     AV取件准备就绪:V512.4
EU
O      INIT:M1.7
NOT
A      AV夹具还原:V512.3
OLD
=      AV夹具还原:V512.3
Network 36
LD     AV1全部放松:V501.7
A      AV2全部放松:V503.7
LD     AV有件:V510.6
O      HMI_RUN_FREE:M1.2
ALD
A      BP_AUTO:I0.5
A      R2_工位1:I7.6
A      AV夹具还原:V512.3
AN     R1_抓件中:M16.0
EU
LD     BP_MANUAL:I0.4
ON     AV1全部放松:V501.7
ON     AV2全部放松:V503.7
LDN    HMI_RUN_FREE:M1.2
AN     AV有件:V510.6
OLD
LD     AV取件:V512.5
EU
OLD
NOT
A      AV取件准备就绪:V512.4
OLD
=      AV取件准备就绪:V512.4
Network 37
LD     R1_IN_JOB2:I5.3
EU
A      AV取件准备就绪:V512.4
A      AV2全部放松:V503.7
A      AV1全部放松:V501.7
A      R1_STAT1_OK:Q4.6
A      R1_AUTO:I5.0
LD     AV取件完成:V512.6
EU
NOT
A      AV取件:V512.5
OLD
=      AV取件:V512.5
Network 38
LD     R1_FINISH2:I6.1
EU
A      AV取件:V512.5
A      R1_AUTO:I5.0
LD     AV全部放松:V510.2
EU
A      AV取件完成:V512.6
NOT
A      AV取件完成:V512.6
OLD
=      AV取件完成:V512.6
END_SUBROUTINE_BLOCK

SUBROUTINE_BLOCK BV:SBR10
TITLE=子程序注释
BEGIN
Network 1 // 网络标题
// 网络注释
LD     BV1全部夹紧:V600.7
A      BV2全部夹紧:V602.7
A      BV3全部夹紧:V604.7
=      BV全部夹紧:V610.1
Network 2
LD     BV1全部放松:V601.7
A      BV2全部放松:V603.7
A      BV3全部放松:V605.7
=      BV全部放松:V610.2
Network 3
LD     BS1:I3.4
A      BS3:I4.6
=      BV有小件:V610.4
Network 4
LD     BS2:I3.5
=      BV有大件:V610.5
Network 5
LD     BV有小件:V610.4
A      BV有大件:V610.5
=      BV有件:V610.6
Network 6
LDN    BS1:I3.4
AN     BS2:I3.5
AN     BS3:I4.6
=      BV未装件:V610.7
Network 7
LDW=   B_JOB_NUM:VW614, +2
OW=    B_JOB_NUM:VW614, +3
=      B工件合格:M14.4
Network 8
LDW=   VW620, +1
OW=    VW620, +4
=      B工件不合格:M14.5
Network 9
LDW=   VW620, +2
OW=    VW620, +3
=      B检测合格:M14.6
Network 10
LDW=   B_JOB_NUM:VW614, +2
=      BV大件偏短:V608.0
Network 11
LDW=   B_JOB_NUM:VW614, +3
=      BV大件偏长:V608.1
Network 12
LDW=   VW616, +2
=      BV焊接偏短:V608.2
Network 13
LDW=   VW616, +3
=      BV焊接偏长:V608.3
Network 14
LDW=   VW618, +2
=      BV取件偏短:V608.4
Network 15
LDW=   VW618, +3
=      BV取件偏长:V608.5
Network 16
LD     B工件不合格:M14.5
A      BP_AUTO:I0.5
R      B1合格组信号1:M11.4, 2
S      B1合格组信号1:M11.4, 1
Network 17
LD     BV大件偏短:V608.0
O      BV取件偏短:V608.4
A      BP_AUTO:I0.5
R      B1合格组信号1:M11.4, 2
S      B1合格组信号2:M11.5, 1
Network 18
LD     BV大件偏长:V608.1
O      BV取件偏长:V608.5
O      B检测合格:M14.6
A      BP_AUTO:I0.5
S      B1合格组信号1:M11.4, 2
Network 19
LD     BP_MANUAL:I0.4
O      BV放大件完成:V611.6
O      BV取件完成:V612.6
ON     CS4:I1.7
R      B1合格组信号1:M11.4, 2
Network 20
LD     BV焊接偏短:V608.2
A      BP_AUTO:I0.5
R      B2合格组信号1:M11.6, 2
S      B2合格组信号2:M11.7, 1
Network 21
LD     BV焊接偏长:V608.3
A      BP_AUTO:I0.5
S      B2合格组信号1:M11.6, 2
Network 22
LD     BP_MANUAL:I0.4
O      BV焊接完成:V612.1
R      B2合格组信号1:M11.6, 2
Network 23
LD     BV全部放松:V610.2
EU
A      BV取件完成:V612.6
AN     ST2_PASS:M2.6
MOVW   +0, VW612
MOVW   +0, VW611
Network 24 // 网络标题
// 网络注释
LD     BV全部放松:V610.2
A      BV未装件:V610.7
LDN    ST1_PASS:M2.4
A      AV焊接完成:V512.1
AN     FINISH:M3.3
LD     开始工作:M0.0
A      ST1_PASS:M2.4
OLD
LDN    FINISH:M3.3
A      R1_HOME:I5.4
A      ST1_PASS:M2.4
OLD
ALD
A      BP_AUTO:I0.5
LDN    HMI_RUN_FREE:M1.2
A      DSL1:I2.2
A      DSR1:I2.6
LD     HMI_RUN_FREE:M1.2
AN     DSL1:I2.2
AN     DSR1:I2.6
OLD
ALD
AW=    VW611, +0
EU
A      R2_工位2:I7.7
LD     BP_MANUAL:I0.4
ON     BV全部放松:V610.2
ON     BV未装件:V610.7
LDN    HMI_RUN_FREE:M1.2
LDN    DSL1:I2.2
ON     DSR1:I2.6
ALD
OLD
LD     HMI_RUN_FREE:M1.2
LD     DSL1:I2.2
O      DSR1:I2.6
ALD
OLD
LD     BV放小件:V611.1
EU
OLD
NOT
A      BV放小件准备就绪:V611.0
OLD
=      BV放小件准备就绪:V611.0
Network 25
LD     R2_IN_JOB1:I7.2
EU
A      BV放小件准备就绪:V611.0
A      R2_AUTO:I7.0
LDW<>  VW511, +0
AN     ST1_PASS:M2.4
A      AV还原准备:V512.2
OW=    VW511, +0
O      ST1_PASS:M2.4
A      BV放小件完成:V611.3
EU
NOT
A      BV放小件:V611.1
OLD
=      BV放小件:V611.1
Network 26
LD     B请求夹紧:I4.7
EU
A      R2_AUTO:I7.0
A      BV放小件:V611.1
LD     BV放小件完成:V611.3
EU
NOT
A      BV请求夹紧:V611.2
OLD
=      BV请求夹紧:V611.2
Network 27
LD     R2_FINISH1:I8.0
EU
A      BV放小件:V611.1
A      R2_AUTO:I7.0
LD     BV放大件:V611.5
EU
NOT
A      BV放小件完成:V611.3
OLD
=      BV放小件完成:V611.3
Network 28
LD     BV放小件完成:V611.3
A      BV1全部放松:V601.7
A      BV2全部夹紧:V602.7
A      BV3全部放松:V605.7
LD     BV有小件:V610.4
O      HMI_RUN_FREE:M1.2
ALD
A      R1_抓件完成:M16.1
AN     BV有大件:V610.5
A      BP_AUTO:I0.5
EU
A      R2_工位2:I7.7
LD     BP_MANUAL:I0.4
ON     BV1全部放松:V601.7
ON     BV2全部夹紧:V602.7
ON     BV3全部放松:V605.7
LDN    HMI_RUN_FREE:M1.2
LDN    BV有小件:V610.4
O      BS2:I3.5
ALD
OLD
LD     BV放大件:V611.5
EU
OLD
NOT
A      BV放大件准备就绪:V611.4
OLD
=      BV放大件准备就绪:V611.4
Network 29
LD     R1_IN_JOB1:I5.2
EU
A      BV放大件准备就绪:V611.4
A      R1_AUTO:I5.0
LD     BV放大件完成:V611.6
EU
NOT
A      BV放大件:V611.5
OLD
=      BV放大件:V611.5
Network 30
LD     BV放大件:V611.5
EU
A      R2_AUTO:I7.0
AW<>   VW511, +0
AN     ST1_PASS:M2.4
LD     AV夹具还原:V512.3
EU
NOT
A      AV还原准备:V512.2
OLD
=      AV还原准备:V512.2
Network 31
LD     R1_FINISH1:I6.0
EU
A      BV放大件:V611.5
A      R1_AUTO:I5.0
LD     BV焊接准备就绪:V611.7
EU
NOT
A      BV放大件完成:V611.6
OLD
=      BV放大件完成:V611.6
Network 32
LD     BV全部夹紧:V610.1
LD     BV有件:V610.6
O      HMI_RUN_FREE:M1.2
ALD
EU
A      BP_AUTO:I0.5
A      R2_工位2:I7.7
A      R2_IN_SAFE:M17.0
LDN    BV全部夹紧:V610.1
LDN    HMI_RUN_FREE:M1.2
AN     BV有件:V610.6
OLD
LD     BV焊接:V612.0
EU
OLD
NOT
A      BV焊接准备就绪:V611.7
OLD
=      BV焊接准备就绪:V611.7
Network 33
LD     R2_IN_JOB2:I7.3
EU
A      BV焊接准备就绪:V611.7
A      R2_AUTO:I7.0
LD     BV焊接完成:V612.1
EU
NOT
A      BV焊接:V612.0
OLD
=      BV焊接:V612.0
Network 34
LD     R2_FINISH2:I8.1
EU
A      BV焊接:V612.0
A      R2_AUTO:I7.0
LD     BV夹具还原:V612.3
EU
NOT
A      BV焊接完成:V612.1
OLD
=      BV焊接完成:V612.1
Network 35
LDN    ST1_PASS:M2.4
A      BV还原准备:V612.2
A      R2_工位2:I7.7
LDN    ST1_PASS:M2.4
A      FINISH:M3.3
A      R2_工位2:I7.7
OLD
O      ST1_PASS:M2.4
A      BV焊接完成:V612.1
EU
A      BP_AUTO:I0.5
LD     BV取件准备就绪:V612.4
EU
NOT
A      BV夹具还原:V612.3
OLD
=      BV夹具还原:V612.3
Network 36
LD     BV1全部放松:V601.7
A      BV2全部放松:V603.7
LD     BV有件:V610.6
O      HMI_RUN_FREE:M1.2
ALD
A      BP_AUTO:I0.5
A      R2_工位2:I7.7
A      BV夹具还原:V612.3
AN     R1_抓件中:M16.0
EU
LD     BP_MANUAL:I0.4
ON     BV1全部放松:V601.7
ON     BV2全部放松:V603.7
LDN    HMI_RUN_FREE:M1.2
AN     BV有件:V610.6
OLD
LD     BV取件:V612.5
EU
OLD
NOT
A      BV取件准备就绪:V612.4
OLD
=      BV取件准备就绪:V612.4
Network 37
LD     R1_IN_JOB2:I5.3
EU
A      BV取件准备就绪:V612.4
A      BV1全部放松:V601.7
A      BV2全部放松:V603.7
A      R1_AUTO:I5.0
LD     BV取件完成:V612.6
EU
NOT
A      BV取件:V612.5
OLD
=      BV取件:V612.5
Network 38
LD     R1_FINISH2:I6.1
EU
A      BV取件:V612.5
A      R1_AUTO:I5.0
LD     BV全部放松:V610.2
EU
A      BV取件完成:V612.6
NOT
A      BV取件完成:V612.6
OLD
=      BV取件完成:V612.6
Network 55 // 网络标题
// 网络注释
END_SUBROUTINE_BLOCK

// SBR11: protected block, not included

// SBR12: protected block, not included

// SBR13: protected block, not included

// SBR14: protected block, not included

// SBR15: protected block, not included

// SBR16: protected block, not included

// SBR17: protected block, not included

// SBR18: protected block, not included

// SBR19: protected block, not included

// SBR20: protected block, not included

// SBR21: protected block, not included

SUBROUTINE_BLOCK 组信号:SBR22
TITLE=子程序注释
BEGIN
Network 1
LD     SM0.1
O      INIT:M1.7
LPS
MOVW   +0, A_JOB_NUM:VW514
AENO
MOVW   +0, VW516
AENO
MOVW   +0, VW518
AENO
MOVW   +0, VW520
LPP
MOVW   +0, B_JOB_NUM:VW614
AENO
MOVW   +0, VW616
AENO
MOVW   +0, VW618
AENO
MOVW   +0, VW620
Network 2
LD     CV2_A:I9.7
EU
LDW>=  T100, +150
ON     CV2_A:I9.7
NOT
A      传送检测气缸信号上:V530.0
OLD
=      传送检测气缸信号上:V530.0
Network 3
LD     CS1:I1.4
EU
LDN    CS1:I1.4
NOT
A      检测CS1:V530.1
OLD
=      检测CS1:V530.1
Network 4
LD     CS3:I1.6
EU
LDN    CV2_A:I9.7
NOT
A      检测CS3:V530.3
OLD
=      检测CS3:V530.3
Network 5
LD     传送检测气缸信号上:V530.0
TON    T100, +200
Network 7
// 偏短,不合格=1
LD     传送检测气缸信号上:V530.0
AN     CS2:I1.5
AN     CS3:I1.6
AW>=   T100, +120
A      SM0.0
MOVW   +1, VW520
MOVW   +1, VW620
Network 8
// 合格，在偏差范围内
LD     传送检测气缸信号上:V530.0
A      CS3:I1.6
AN     CS2:I1.5
AW>=   T100, +120
A      SM0.0
MOVW   +2, VW520
MOVW   +2, VW620
Network 9
LD     传送检测气缸信号上:V530.0
A      CS1:I1.4
A      CS2:I1.5
AN     CS3:I1.6
AW>=   T100, +120
AN     SM0.0
A      SM0.0
LD     HMI_RUN_FREE:M1.2
AN     CS4:I1.7
AN     CS1:I1.4
AN     CS2:I1.5
AN     CS3:I1.6
A      SM0.0
OLD
MOVW   +3, VW520
MOVW   +3, VW620
Network 10
// 不合格,偏长=4
LD     传送检测气缸信号上:V530.0
A      CS2:I1.5
A      CS3:I1.6
AW>=   T100, +120
A      SM0.0
MOVW   +4, VW520
MOVW   +4, VW620
Network 11
LDW>=  T100, +120
AN     CS3:I1.6
A      CS2:I1.5
LDW>=  T100, +120
AN     CS1:I1.4
A      CS2:I1.5
A      CS3:I1.6
AN     SM0.0
OLD
LDW>=  T100, +120
AN     CS1:I1.4
AN     CS2:I1.5
A      CS3:I1.6
AN     SM0.0
OLD
LDW>=  T100, +120
AN     CS1:I1.4
A      CS2:I1.5
AN     CS3:I1.6
AN     SM0.0
OLD
MOVW   +0, VW520
MOVW   +0, VW620
Network 12
// 虚拟
LD     SM0.1
R      虚拟:M31.2, 1
Network 13
// 虚拟
LD     BP_DOOR_RESET1:I1.3
TON    T150, +20
Network 14
// 虚拟
LD     T150
R      虚拟:M31.2, 1
Network 15
// 虚拟
LD     BP_DOOR_RESET1:I1.3
EU
S      虚拟:M31.2, 1
Network 16
LD     BP_DOOR_RESET1:I1.3
EU
AN     虚拟reset:M31.3
LD     BP_DOOR_RESET1:I1.3
EU
A      虚拟reset:M31.3
NOT
A      虚拟:M31.2
OLD
=      虚拟:M31.2
Network 17
LD     BP_DOOR_RESET1:I1.3
ED
A      虚拟:M31.2
LD     BP_DOOR_RESET1:I1.3
ED
AN     虚拟:M31.2
NOT
A      虚拟reset:M31.3
OLD
=      虚拟reset:M31.3
Network 18
// 虚拟
LD     虚拟:M31.2
LD     CS4:I1.7
O      HMI_RUN_FREE:M1.2
ALD
MOVW   +3, VW520
MOVW   +3, VW620
Network 19
LDN    HMI_RUN_FREE:M1.2
AN     CS4:I1.7
MOVW   +0, VW520
MOVW   +0, VW620
Network 20
LD     SM0.0
LPS
A      AV放大件准备就绪:V511.4
EU
AN     SM0.0
MOVW   VW520, A_JOB_NUM:VW514
AENO
MOVW   +0, VW520
LPP
A      BV放大件准备就绪:V611.4
EU
AN     SM0.0
MOVW   VW620, B_JOB_NUM:VW614
AENO
MOVW   +0, VW620
Network 21
LD     AV放大件完成:V511.6
EU
AN     SM0.0
MOVW   A_JOB_NUM:VW514, VW516
AENO
MOVW   +0, A_JOB_NUM:VW514
Network 22
LD     AV焊接完成:V512.1
EU
AN     SM0.0
MOVW   VW516, VW518
AENO
MOVW   +0, VW516
Network 23
LD     AV取件完成:V512.6
EU
MOVW   +0, VW518
Network 24
LD     SM0.0
MOVW   +0, A_JOB_NUM:VW514
AENO
MOVW   +0, VW516
AENO
MOVW   +0, VW518
Network 25
LD     BV放大件完成:V611.6
EU
AN     SM0.0
MOVW   B_JOB_NUM:VW614, VW616
AENO
MOVW   +0, B_JOB_NUM:VW614
Network 26
LD     BV焊接完成:V612.1
EU
AN     SM0.0
MOVW   VW616, VW618
AENO
MOVW   +0, VW616
Network 27
LD     BV取件完成:V612.6
EU
MOVW   +0, VW618
Network 28
LD     SM0.0
MOVW   +0, B_JOB_NUM:VW614
AENO
MOVW   +0, VW616
AENO
MOVW   +0, VW618
END_SUBROUTINE_BLOCK

SUBROUTINE_BLOCK PLC_ROBOT1:SBR23
TITLE=子程序注释
BEGIN
Network 1
LD     R1_HOME:I5.4
=      R1_IN_SAFE:M15.0
Network 2
// 复位机器人的急停
LD     BP_ES_RESET:I0.2
A      R1_AUTO:I5.0
TON    T50, +20
Network 3
LD     T50
=      R1_RESET_ES:Q4.3
Network 4 // 网络标题
LD     ATUOSTART:M10.2
A      R1_AUTO:I5.0
A      R1_START:M15.1
=      RI_CYCLE_START:Q4.1
Network 5
// 从FIXTURE 回 HOME
LDN    ATUOSTART:M10.2
A      R1_CYCLE_NO:I5.1
A      R1_HOME:I5.4
LD     ST1_WORKING:M3.0
O      ST2_WORKING:M3.1
A      PAUSE:M2.3
A      R1_AUTO:I5.0
A      R1_CYCLE_NO:I5.1
OLD
=      R1_CYCLE_STOP:Q4.2
Network 6
LD     ATUOSTART:M10.2
LD     R1_AUTO:I5.0
O      R1_IN_SAFE:M15.0
ALD
LDN    R1_AUTO:I5.0
NOT
A      R1_START:M15.1
OLD
=      R1_START:M15.1
Network 7
// 启动机器人的系统程序
LD     ATUOSTART:M10.2
A      R1_IN_SAFE:M15.0
EU
LD     WORK_START:I0.1
AN     PAUSE:M2.3
EU
LD     ST1_WORKING:M3.0
O      ST2_WORKING:M3.1
ALD
OLD
LD     R1_CYCLE_NO:I5.1
NOT
A      R1_PRO_START:Q4.0
OLD
=      R1_PRO_START:Q4.0
Network 8
// 机器人启动就绪,等待工作
LD     R1_AUTO:I5.0
A      R1_CYCLE_NO:I5.1
A      R1_IN_SAFE:M15.0
A      ES_OK:I0.7
A      AS_OK:I1.2
AN     R1_IN_JOB1:I5.2
AN     R1_IN_JOB2:I5.3
=      R1_JOB_READY:M15.4
Network 9
LD     AV放大件准备就绪:V511.4
O      AV取件准备就绪:V512.4
A      BP_AUTO:I0.5
A      R1_AUTO:I5.0
A      R1_CYCLE_NO:I5.1
A      R2_工位1:I7.6
AN     R1_IN_JOB1:I5.2
AN     R1_IN_JOB2:I5.3
A      R1_IN_SAFE:M15.0
AN     R1_STAT2_OK:Q4.7
=      R1_STAT1_OK:Q4.6
Network 10
LD     BV放大件准备就绪:V611.4
O      BV取件准备就绪:V612.4
A      BP_AUTO:I0.5
A      R1_AUTO:I5.0
A      R1_CYCLE_NO:I5.1
A      R2_工位2:I7.7
A      R1_IN_SAFE:M15.0
AN     R1_IN_JOB1:I5.2
AN     R1_IN_JOB2:I5.3
AN     R1_STAT1_OK:Q4.6
=      R1_STAT2_OK:Q4.7
Network 11
// 产品组信号1
LD     R1_AUTO:I5.0
A      R1_CYCLE_NO:I5.1
A      BP_AUTO:I0.5
LDN    R1_AUTO:I5.0
A      BP_MANUAL:I0.4
OLD
A      产品组信号1:M12.0
=      R1_POS1:Q5.2
Network 12
LD     R1_AUTO:I5.0
A      R1_CYCLE_NO:I5.1
A      BP_AUTO:I0.5
LDN    R1_AUTO:I5.0
A      BP_MANUAL:I0.4
OLD
A      产品组信号2:M12.1
=      R1_POS2:Q5.3
Network 13
LD     R1_AUTO:I5.0
A      R1_CYCLE_NO:I5.1
A      BP_AUTO:I0.5
LDN    R1_AUTO:I5.0
A      BP_MANUAL:I0.4
OLD
A      产品组信号3:M12.2
=      R1_POS3:Q5.4
Network 14
LD     R1_AUTO:I5.0
A      R1_CYCLE_NO:I5.1
A      BP_AUTO:I0.5
LDN    R1_AUTO:I5.0
A      BP_MANUAL:I0.4
OLD
A      产品组信号4:M12.3
=      R1_POS4:Q5.5
Network 15
LD     SM0.0
MOVB   QB5, VB800
AENO
SLB    VB800, 2
AENO
MOVB   VB800, VB801
SRB    VB801, 4
Network 16
LD     SM0.0
MOVB   IB6, VB802
AENO
SLB    VB802, 2
AENO
MOVB   VB802, VB803
SRB    VB803, 4
Network 17
LDB=   VB801, VB803
AB<>   VB801, 0
=      R1_POS_OK:M15.5
Network 18
LD     A1合格组信号1:M11.0
O      B1合格组信号1:M11.4
A      BP_AUTO:I0.5
A      ES_OK:I0.7
A      AS_OK:I1.2
A      R1_AUTO:I5.0
A      R1_CYCLE_NO:I5.1
AN     CV2_A:I9.7
AN     R1_抓件中:M16.0
=      R1_PIC1:Q5.6
Network 19
LD     A1合格组信号2:M11.1
O      B1合格组信号2:M11.5
A      BP_AUTO:I0.5
A      ES_OK:I0.7
A      AS_OK:I1.2
A      R1_AUTO:I5.0
A      R1_CYCLE_NO:I5.1
AN     CV2_A:I9.7
AN     R1_抓件中:M16.0
=      R1_PIC2:Q5.7
Network 20
LD     R1_PIC1:Q5.6
AN     R1_PIC2:Q5.7
A      IN_R1_PIC1:I6.6
AN     IN_R1_PIC2:I6.7
LDN    R1_PIC1:Q5.6
A      R1_PIC2:Q5.7
AN     IN_R1_PIC1:I6.6
A      IN_R1_PIC2:I6.7
OLD
LD     R1_PIC1:Q5.6
A      R1_PIC2:Q5.7
A      IN_R1_PIC1:I6.6
A      IN_R1_PIC2:I6.7
OLD
=      R1_PIC_OK:M15.6
Network 21
LD     AV放小件准备就绪:V511.0
O      AV放小件:V511.1
O      AV请求夹紧:V511.2
O      AV放小件完成:V511.3
AN     ST1_PASS:M2.4
A      A检测合格:M14.2
=      AV允许抓大件:M4.0
Network 22
LD     BV放小件准备就绪:V611.0
O      BV放小件:V611.1
O      BV请求夹紧:V611.2
O      BV放小件完成:V611.3
AN     ST2_PASS:M2.6
A      B检测合格:M14.6
=      BV允许抓大件:M4.1
Network 23
LD     AV允许抓大件:M4.0
O      BV允许抓大件:M4.1
A      BP_AUTO:I0.5
A      ES_OK:I0.7
A      AS_OK:I1.2
A      R1_AUTO:I5.0
A      R1_CYCLE_NO:I5.1
AN     R1_抓件中:M16.0
A      R1_HOME:I5.4
AN     R1_UNLOAD_OK:Q5.0
AN     CV2_A:I9.7
S      R1_UNLOAD_OK:Q5.0, 1
Network 24
LDN    BP_AUTO:I0.5
O      INIT:M1.7
O      R1_抓件中:M16.0
O      CV2_A:I9.7
O      R1_抓件完成:M16.1
R      R1_UNLOAD_OK:Q5.0, 1
Network 25
LD     R1_PIC_OK:M15.6
A      R1_POS_OK:M15.5
A      BP_AUTO:I0.5
A      ES_OK:I0.7
AN     R1_抓件中:M16.0
A      AS_OK:I1.2
A      R1_AUTO:I5.0
A      R1_CYCLE_NO:I5.1
A      R1_HOME:I5.4
=      R1_JOB3_VALD:Q5.1
Network 26
LD     R1_IN_UNLOAD:I5.6
EU
LD     AV放大件:V511.5
EU
LD     BV放大件:V611.5
EU
OLD
O      INIT:M1.7
NOT
A      R1_抓件中:M16.0
OLD
=      R1_抓件中:M16.0
Network 27
LD     R1_FINISH3:I5.7
EU
LD     AV放大件:V511.5
EU
LD     BV放大件:V611.5
EU
OLD
O      INIT:M1.7
NOT
A      R1_抓件完成:M16.1
OLD
=      R1_抓件完成:M16.1
Network 28
// 机器人1开始放件
LD     AV放大件准备就绪:V511.4
A      R2_IN_SAFE:M17.0
A      R2_工位1:I7.6
A      R1_STAT1_OK:Q4.6
LD     BV放大件准备就绪:V611.4
A      R2_IN_SAFE:M17.0
A      R2_工位2:I7.7
A      R1_STAT2_OK:Q4.7
OLD
A      R1_JOB_READY:M15.4
A      R1_POS_OK:M15.5
=      R1_JOB1_VAILD:Q4.4
Network 29
LD     AV取件准备就绪:V512.4
A      R1_STAT1_OK:Q4.6
LD     BV取件准备就绪:V612.4
A      R1_STAT2_OK:Q4.7
OLD
A      R1_JOB_READY:M15.4
A      R1_POS_OK:M15.5
=      R1_JOB2_VAILD:Q4.5
END_SUBROUTINE_BLOCK

SUBROUTINE_BLOCK PLC_ROBOT2:SBR24
TITLE=子程序注释
BEGIN
Network 1
LD     R2_HOME:I7.4
=      R2_IN_SAFE:M17.0
Network 2
// 复位机器人的急停
LD     BP_ES_RESET:I0.2
A      R2_AUTO:I7.0
TON    T60, +20
Network 3
LD     T60
=      R2_RESET_ES:Q6.3
Network 4 // 网络标题
LD     ATUOSTART:M10.2
A      R2_AUTO:I7.0
A      R2_START:M17.1
=      R2_CYCLE_START:Q6.1
Network 5
// 从FIXTURE 回 HOME
LDN    ATUOSTART:M10.2
A      R2_CYCLE_NO:I7.1
A      R2_HOME:I7.4
LD     ST1_WORKING:M3.0
O      ST2_WORKING:M3.1
A      PAUSE:M2.3
A      R2_AUTO:I7.0
A      R2_CYCLE_NO:I7.1
OLD
=      R2_CYCLE_STOP:Q6.2
Network 6
LD     ATUOSTART:M10.2
LD     R2_AUTO:I7.0
O      R2_IN_SAFE:M17.0
ALD
LDN    R2_AUTO:I7.0
NOT
A      R2_START:M17.1
OLD
=      R2_START:M17.1
Network 7
// 启动机器人的系统程序
LD     ATUOSTART:M10.2
A      R2_IN_SAFE:M17.0
EU
LD     WORK_START:I0.1
AN     PAUSE:M2.3
EU
LD     ST1_WORKING:M3.0
O      ST2_WORKING:M3.1
ALD
OLD
LD     R2_CYCLE_NO:I7.1
NOT
A      R2_PRO_START:Q6.0
OLD
=      R2_PRO_START:Q6.0
Network 8
// 机器人启动就绪,等待工作
LD     R2_AUTO:I7.0
A      R2_CYCLE_NO:I7.1
A      R2_IN_SAFE:M17.0
LD     R2_工位1:I7.6
O      R2_工位2:I7.7
ALD
A      ES_OK:I0.7
A      AS_OK:I1.2
AN     R2_IN_JOB1:I7.2
AN     R2_IN_JOB2:I7.3
=      R2_JOB_READY:M17.4
Network 9
LD     AV放小件准备就绪:V511.0
O      AV焊接准备就绪:V511.7
A      R2_AUTO:I7.0
A      R2_CYCLE_NO:I7.1
A      BP_AUTO:I0.5
A      R2_工位1:I7.6
A      R2_IN_SAFE:M17.0
AN     R2_IN_JOB1:I7.2
AN     R2_IN_JOB2:I7.3
AN     R2_STAT2_OK:Q6.7
=      R2_STAT1_OK:Q6.6
Network 10
LD     BV放小件准备就绪:V611.0
O      BV焊接准备就绪:V611.7
A      R2_AUTO:I7.0
A      R2_CYCLE_NO:I7.1
A      BP_AUTO:I0.5
A      R2_工位2:I7.7
A      R2_IN_SAFE:M17.0
AN     R2_IN_JOB1:I7.2
AN     R2_IN_JOB2:I7.3
AN     R2_STAT1_OK:Q6.6
=      R2_STAT2_OK:Q6.7
Network 11
// 产品组信号1
LD     R2_AUTO:I7.0
A      R2_CYCLE_NO:I7.1
A      BP_AUTO:I0.5
LD     R2_STAT1_OK:Q6.6
AN     R2_STAT2_OK:Q6.7
LDN    R2_STAT1_OK:Q6.6
A      R2_STAT2_OK:Q6.7
OLD
ALD
LDN    R2_AUTO:I7.0
A      BP_MANUAL:I0.4
OLD
A      产品组信号1:M12.0
=      R2_POS1:Q7.2
Network 12
LD     R2_AUTO:I7.0
A      R2_CYCLE_NO:I7.1
A      BP_AUTO:I0.5
LD     R2_STAT1_OK:Q6.6
AN     R2_STAT2_OK:Q6.7
LDN    R2_STAT1_OK:Q6.6
A      R2_STAT2_OK:Q6.7
OLD
ALD
LDN    R2_AUTO:I7.0
A      BP_MANUAL:I0.4
OLD
A      产品组信号2:M12.1
=      R2_POS2:Q7.3
Network 13
LD     R2_AUTO:I7.0
A      R2_CYCLE_NO:I7.1
A      BP_AUTO:I0.5
LD     R2_STAT1_OK:Q6.6
AN     R2_STAT2_OK:Q6.7
LDN    R2_STAT1_OK:Q6.6
A      R2_STAT2_OK:Q6.7
OLD
ALD
LDN    R2_AUTO:I7.0
A      BP_MANUAL:I0.4
OLD
A      产品组信号3:M12.2
=      R2_POS3:Q7.4
Network 14
LD     R2_AUTO:I7.0
A      R2_CYCLE_NO:I7.1
A      BP_AUTO:I0.5
LD     R2_STAT1_OK:Q6.6
AN     R2_STAT2_OK:Q6.7
LDN    R2_STAT1_OK:Q6.6
A      R2_STAT2_OK:Q6.7
OLD
ALD
LDN    R2_AUTO:I7.0
A      BP_MANUAL:I0.4
OLD
A      产品组信号4:M12.3
=      R2_POS4:Q7.5
Network 15
LD     SM0.0
MOVB   QB7, VB810
AENO
SLB    VB810, 2
AENO
MOVB   VB810, VB811
SRB    VB811, 4
Network 16
LD     SM0.0
MOVB   IB8, VB812
AENO
SLB    VB812, 2
AENO
MOVB   VB812, VB813
SRB    VB813, 4
Network 17
LDB=   VB811, VB813
AB<>   VB811, 0
=      R2_POS_OK:M17.5
Network 18
LD     A2合格组信号1:M11.2
O      B2合格组信号1:M11.6
A      BP_AUTO:I0.5
A      ES_OK:I0.7
A      AS_OK:I1.2
A      R2_AUTO:I7.0
A      R2_CYCLE_NO:I7.1
=      R2_PIC1:Q7.6
Network 19
LD     A2合格组信号2:M11.3
O      B2合格组信号2:M11.7
A      BP_AUTO:I0.5
A      ES_OK:I0.7
A      AS_OK:I1.2
A      R2_AUTO:I7.0
A      R2_CYCLE_NO:I7.1
=      R2_PIC2:Q7.7
Network 20
LD     R2_PIC1:Q7.6
AN     R2_PIC2:Q7.7
A      IN_R2_PIC1:I8.6
AN     IN_R2_PIC2:I8.7
LDN    R2_PIC1:Q7.6
A      R2_PIC2:Q7.7
AN     IN_R2_PIC1:I8.6
A      IN_R2_PIC2:I8.7
OLD
LD     R2_PIC1:Q7.6
A      R2_PIC2:Q7.7
A      IN_R2_PIC1:I8.6
A      IN_R2_PIC2:I8.7
OLD
=      R2_PIC_OK:M17.6
Network 21
// 机器人2开始抓件
LD     AV未装件:V510.7
A      AV放小件准备就绪:V511.0
A      R2_工位1:I7.6
A      R2_STAT1_OK:Q6.6
LD     BV未装件:V610.7
A      BV放小件准备就绪:V611.0
A      R2_工位2:I7.7
A      R2_STAT2_OK:Q6.7
OLD
A      R2_JOB_READY:M17.4
A      R2_POS_OK:M17.5
=      R2_JOB1_VAILD:Q6.4
Network 22
// 机器人2开始焊接
LD     AV焊接准备就绪:V511.7
A      AV全部夹紧:V510.1
LD     AV有件:V510.6
O      HMI_RUN_FREE:M1.2
ALD
A      R2_IN_SAFE:M17.0
A      R2_工位1:I7.6
A      R2_STAT1_OK:Q6.6
LD     BV焊接准备就绪:V611.7
A      BV全部夹紧:V610.1
LD     BV有件:V610.6
O      HMI_RUN_FREE:M1.2
ALD
A      R2_IN_SAFE:M17.0
A      R2_工位2:I7.7
A      R2_STAT2_OK:Q6.7
OLD
A      R2_JOB_READY:M17.4
A      R2_POS_OK:M17.5
=      R2_JOB2_VAILD:Q6.5
Network 23
LD     A请求夹紧:I3.7
A      AV2全部夹紧:V502.7
A      R2_AUTO:I7.0
A      BP_AUTO:I0.5
=      R2_A_小件夹紧:Q7.0
Network 24
LD     B请求夹紧:I4.7
A      BV2全部夹紧:V602.7
A      R2_AUTO:I7.0
A      BP_AUTO:I0.5
=      R2_B_小件夹紧:Q7.1
END_SUBROUTINE_BLOCK

SUBROUTINE_BLOCK SBR_25:SBR25
TITLE=子程序注释
VAR_INPUT
EIN:BOOL;	// L0.0 
LENGTH:INT;	// LW1 
END_VAR
VAR
TEMP1:WORD;	// LW3 
TEMP2:DWORD;	// LD5 
TEMP3:DWORD;	// LD9 
TEMP10:WORD;	// LW13 
TEMP11:WORD;	// LW15 
TEMP12:WORD;	// LW17 
TEMP13:WORD;	// LW19 
END_VAR
BEGIN
Network 1 // 网络标题
// 网络注释
LD     #EIN:L0.0
ON     #EIN:L0.0
=      #EIN:L0.0
Network 2
LD     SM0.1
MOVW   +1, #TEMP1:LW3
MOVD   +0, #TEMP2:LD5
MOVD   +0, #TEMP3:LD9
Network 3
LD     #EIN:L0.0
MOVD   &VB400, #TEMP2:LD5
MOVD   &VB700, #TEMP3:LD9
Network 4
LD     #EIN:L0.0
FOR    #TEMP1:LW3, +1, #LENGTH:LW1
Network 6
LD     #EIN:L0.0
MOVW   *#TEMP2:LD5, #TEMP10:LW13
Network 7
LD     #EIN:L0.0
MOVW   #TEMP10:LW13, #TEMP11:LW15
AENO
SLW    #TEMP11:LW15, 8
AENO
MOVW   #TEMP10:LW13, #TEMP12:LW17
SRW    #TEMP12:LW17, 8
Network 8
LD     #EIN:L0.0
MOVW   #TEMP11:LW15, #TEMP13:LW19
AENO
ORW    #TEMP12:LW17, #TEMP13:LW19
AENO
MOVW   #TEMP13:LW19, *#TEMP3:LD9
Network 9
LD     #EIN:L0.0
+D     +2, #TEMP2:LD5
+D     +2, #TEMP3:LD9
Network 10
NEXT
END_SUBROUTINE_BLOCK

// SBR26: protected block, not included

// SBR27: protected block, not included

// SBR28: protected block, not included

// SBR29: protected block, not included

// SBR30: protected block, not included

// SBR31: protected block, not included

// SBR32: protected block, not included

// SBR33: protected block, not included

// SBR34: protected block, not included

// SBR35: protected block, not included

// SBR36: protected block, not included

SUBROUTINE_BLOCK MESS_1:SBR37
TITLE=子程序注释
VAR_INPUT
VALVE:BOOL;	// L0.0 
INPUT1:BOOL;	// L0.1 
INPUT2:BOOL;	// L0.2 
INPUT3:BOOL;	// L0.3 
INPUT4:BOOL;	// L0.4 
ACT:BOOL;	// L0.5 
END_VAR
VAR_OUTPUT
MESS1:BOOL;	// L0.6 
MESS2:BOOL;	// L0.7 
MESS3:BOOL;	// L1.0 
MESS4:BOOL;	// L1.1 
RESET:BOOL;	// L1.2 
END_VAR
BEGIN
Network 1
LD     #ACT:L0.5
A      #VALVE:L0.0
AN     #INPUT1:L0.1
=      #MESS1:L0.6
Network 2
LD     #ACT:L0.5
A      #VALVE:L0.0
AN     #INPUT2:L0.2
=      #MESS2:L0.7
Network 3
LD     #ACT:L0.5
A      #VALVE:L0.0
AN     #INPUT3:L0.3
=      #MESS3:L1.0
Network 4
LD     #ACT:L0.5
A      #VALVE:L0.0
AN     #INPUT4:L0.4
=      #MESS4:L1.1
Network 5
LD     #INPUT1:L0.1
A      #INPUT2:L0.2
A      #INPUT3:L0.3
A      #INPUT4:L0.4
=      #RESET:L1.2
END_SUBROUTINE_BLOCK

SUBROUTINE_BLOCK MESS_2:SBR38
TITLE=子程序注释
BEGIN
Network 1
LD     AV1_A:Q8.0
EU
O      AV1_A_RES:V426.0
MOVB   0, VB430
AENO
LD     AV1_B:Q8.1
EU
O      AV1_B_RES:V426.1
MOVB   0, VB431
AENO
OLD
LD     AV2_A:Q8.4
EU
O      AV2_A_RES:V426.2
MOVB   0, VB432
AENO
OLD
LD     AV2_B:Q8.5
EU
O      AV2_B_RES:V426.3
MOVB   0, VB433
AENO
OLD
LD     AV3_A:Q8.6
EU
O      AV3_A_RES:V426.4
MOVB   0, VB434
AENO
OLD
LD     AV3_B:Q8.7
EU
O      AV3_B_RES:V426.5
MOVB   0, VB435
AENO
OLD
=      DUMMY:M31.0
Network 2
LD     BV1_A:Q10.0
EU
O      BV1_A_RES:V427.0
MOVB   0, VB440
AENO
LD     BV1_B:Q10.1
EU
O      BV1_B_RES:V427.1
MOVB   0, VB441
AENO
OLD
LD     BV2_A:Q10.4
EU
O      BV2_A_RES:V427.2
MOVB   0, VB442
AENO
OLD
LD     BV2_B:Q10.5
EU
O      BV2_B_RES:V427.3
MOVB   0, VB443
AENO
OLD
LD     BV3_A:Q10.6
EU
O      BV3_A_RES:V427.4
MOVB   0, VB444
AENO
OLD
LD     BV3_B:Q10.7
EU
O      BV3_B_RES:V427.5
MOVB   0, VB445
AENO
OLD
=      DUMMY:M31.0
Network 3
LD     SM0.5
EU
LPS
A      AV1_A:Q8.0
INCB   VB430
LRD
A      AV1_B:Q8.1
INCB   VB431
LRD
A      AV2_A:Q8.4
INCB   VB432
LRD
A      AV2_B:Q8.5
INCB   VB433
LRD
A      AV3_A:Q8.6
INCB   VB434
LPP
A      AV3_B:Q8.7
INCB   VB435
Network 4
LD     SM0.5
EU
LPS
A      BV1_A:Q10.0
INCB   VB440
LRD
A      BV1_B:Q10.1
INCB   VB441
LRD
A      BV2_A:Q10.4
INCB   VB442
LRD
A      BV2_B:Q10.5
INCB   VB443
LRD
A      BV3_A:Q10.6
INCB   VB444
LPP
A      BV3_B:Q10.7
INCB   VB445
Network 5
LD     SM0.0
LPS
AB>=   VB430, 6
=      AV1_A_CAT:V422.0
LRD
AB>=   VB431, 6
=      AV1_B_CAT:V422.1
LRD
AB>=   VB432, 6
=      AV2_A_CAT:V422.2
LRD
AB>=   VB433, 6
=      AV2_B_CAT:V422.3
LRD
AB>=   VB434, 6
=      AV3_A_CAT:V422.4
LPP
AB>=   VB435, 6
=      AV3_B_CAT:V422.5
Network 6
LD     SM0.0
LPS
AB>=   VB440, 6
=      BV1_A_CAT:V423.0
LRD
AB>=   VB441, 6
=      BV1_B_CAT:V423.1
LRD
AB>=   VB442, 6
=      BV2_A_CAT:V423.2
LRD
AB>=   VB443, 6
=      BV2_B_CAT:V423.3
LRD
AB>=   VB444, 6
=      BV3_A_CAT:V423.4
LPP
AB>=   VB445, 6
=      BV3_B_CAT:V423.5
Network 7
LD     SM0.0
=      L60.0
LD     AV1_A:Q8.0
=      L63.7
LD     AV1_1A:I9.0
=      L63.6
LD     AV1_2A:I9.2
=      L63.5
LD     SM0.0
=      L63.4
LD     SM0.0
=      L63.3
LD     AV1_A_CAT:V422.0
=      L63.2
LD     L60.0
CALL   MESS_1:SBR37, L63.7, L63.6, L63.5, L63.4, L63.3, L63.2, AV1_1A_MESS:V400.0, AV1_2A_MESS:V400.1, AV1_3A_MESS:V400.2, AV1_4A_MESS:V400.3, AV1_A_RES:V426.0
Network 8
LD     SM0.0
=      L60.0
LD     AV1_B:Q8.1
=      L63.7
LD     AV1_1B:I9.1
=      L63.6
LD     AV1_2B:I9.3
=      L63.5
LD     SM0.0
=      L63.4
LD     SM0.0
=      L63.3
LD     AV1_B_CAT:V422.1
=      L63.2
LD     L60.0
CALL   MESS_1:SBR37, L63.7, L63.6, L63.5, L63.4, L63.3, L63.2, AV1_1B_MESS:V400.4, AV1_2B_MESS:V400.5, AV1_3B_MESS:V400.6, AV1_4B_MESS:V400.7, AV1_B_RES:V426.1
Network 9
LD     SM0.0
=      L60.0
LD     AV2_A:Q8.4
=      L63.7
LD     AV2_1A:I10.0
=      L63.6
LD     AV2_2A:I10.2
=      L63.5
LD     SM0.0
=      L63.4
LD     SM0.0
=      L63.3
LD     AV2_A_CAT:V422.2
=      L63.2
LD     L60.0
CALL   MESS_1:SBR37, L63.7, L63.6, L63.5, L63.4, L63.3, L63.2, AV2_1A_MESS:V401.0, AV2_2A_MESS:V401.1, AV2_3A_MESS:V401.2, AV2_4A_MESS:V401.3, AV2_A_RES:V426.2
Network 10
LD     SM0.0
=      L60.0
LD     AV2_B:Q8.5
=      L63.7
LD     AV2_1B:I10.1
=      L63.6
LD     AV2_2B:I10.3
=      L63.5
LD     SM0.0
=      L63.4
LD     SM0.0
=      L63.3
LD     AV2_B_CAT:V422.3
=      L63.2
LD     L60.0
CALL   MESS_1:SBR37, L63.7, L63.6, L63.5, L63.4, L63.3, L63.2, AV2_1B_MESS:V401.4, AV2_2B_MESS:V401.5, AV2_3B_MESS:V401.6, AV2_4B_MESS:V401.7, AV2_B_RES:V426.3
Network 11
LD     SM0.0
=      L60.0
LD     AV3_A:Q8.6
=      L63.7
LD     AV3_1A:I10.4
=      L63.6
LD     SM0.0
=      L63.5
LD     SM0.0
=      L63.4
LD     SM0.0
=      L63.3
LD     AV3_A_CAT:V422.4
=      L63.2
LD     L60.0
CALL   MESS_1:SBR37, L63.7, L63.6, L63.5, L63.4, L63.3, L63.2, AV3_1A_MESS:V402.0, AV3_2A_MESS:V402.1, AV3_3A_MESS:V402.2, AV3_4A_MESS:V402.3, AV3_A_RES:V426.4
Network 12
LD     SM0.0
=      L60.0
LD     AV3_B:Q8.7
=      L63.7
LD     AV3_1B:I10.5
=      L63.6
LD     SM0.0
=      L63.5
LD     SM0.0
=      L63.4
LD     SM0.0
=      L63.3
LD     AV3_B_CAT:V422.5
=      L63.2
LD     L60.0
CALL   MESS_1:SBR37, L63.7, L63.6, L63.5, L63.4, L63.3, L63.2, AV3_1B_MESS:V402.4, AV3_2B_MESS:V402.5, AV3_3B_MESS:V402.6, AV3_4B_MESS:V402.7, AV3_B_RES:V426.5
Network 13
LD     SM0.0
=      L60.0
LD     BV1_A:Q10.0
=      L63.7
LD     BV1_1A:I3.0
=      L63.6
LD     BV1_2A:I3.2
=      L63.5
LD     SM0.0
=      L63.4
LD     SM0.0
=      L63.3
LD     BV1_A_CAT:V423.0
=      L63.2
LD     L60.0
CALL   MESS_1:SBR37, L63.7, L63.6, L63.5, L63.4, L63.3, L63.2, BV1_1A_MESS:V404.0, BV1_2A_MESS:V404.1, BV1_3A_MESS:V404.2, BV1_4A_MESS:V404.3, BV1_A_RES:V427.0
Network 14
LD     SM0.0
=      L60.0
LD     BV1_B:Q10.1
=      L63.7
LD     BV1_1B:I3.1
=      L63.6
LD     BV1_2B:I3.3
=      L63.5
LD     SM0.0
=      L63.4
LD     SM0.0
=      L63.3
LD     BV1_B_CAT:V423.1
=      L63.2
LD     L60.0
CALL   MESS_1:SBR37, L63.7, L63.6, L63.5, L63.4, L63.3, L63.2, BV1_1B_MESS:V404.4, BV1_2B_MESS:V404.5, BV1_3B_MESS:V404.6, BV1_4B_MESS:V404.7, BV1_B_RES:V427.1
Network 15
LD     SM0.0
=      L60.0
LD     BV2_A:Q10.4
=      L63.7
LD     BV2_1A:I4.0
=      L63.6
LD     BV2_2A:I4.2
=      L63.5
LD     SM0.0
=      L63.4
LD     SM0.0
=      L63.3
LD     BV2_A_CAT:V423.2
=      L63.2
LD     L60.0
CALL   MESS_1:SBR37, L63.7, L63.6, L63.5, L63.4, L63.3, L63.2, BV2_1A_MESS:V405.0, BV2_2A_MESS:V405.1, BV2_3A_MESS:V405.2, BV2_4A_MESS:V405.3, BV2_A_RES:V427.2
Network 16
LD     SM0.0
=      L60.0
LD     BV2_B:Q10.5
=      L63.7
LD     BV2_1B:I4.1
=      L63.6
LD     BV2_2B:I4.3
=      L63.5
LD     SM0.0
=      L63.4
LD     SM0.0
=      L63.3
LD     BV2_B_CAT:V423.3
=      L63.2
LD     L60.0
CALL   MESS_1:SBR37, L63.7, L63.6, L63.5, L63.4, L63.3, L63.2, BV2_1B_MESS:V405.4, BV2_2B_MESS:V405.5, BV2_3B_MESS:V405.6, BV2_4B_MESS:V405.7, BV2_B_RES:V427.3
Network 17
LD     SM0.0
=      L60.0
LD     BV3_A:Q10.6
=      L63.7
LD     BV3_1A:I4.4
=      L63.6
LD     SM0.0
=      L63.5
LD     SM0.0
=      L63.4
LD     SM0.0
=      L63.3
LD     BV3_A_CAT:V423.4
=      L63.2
LD     L60.0
CALL   MESS_1:SBR37, L63.7, L63.6, L63.5, L63.4, L63.3, L63.2, BV3_1A_MESS:V406.0, BV3_2A_MESS:V406.1, BV3_3A_MESS:V406.2, BV3_4A_MESS:V406.3, BV3_A_RES:V427.4
Network 18
LD     SM0.0
=      L60.0
LD     BV3_B:Q10.7
=      L63.7
LD     BV3_1B:I4.5
=      L63.6
LD     SM0.0
=      L63.5
LD     SM0.0
=      L63.4
LD     SM0.0
=      L63.3
LD     BV3_B_CAT:V423.5
=      L63.2
LD     L60.0
CALL   MESS_1:SBR37, L63.7, L63.6, L63.5, L63.4, L63.3, L63.2, BV3_1B_MESS:V406.4, BV3_2B_MESS:V406.5, BV3_3B_MESS:V406.6, BV3_4B_MESS:V406.7, BV3_B_RES:V427.5
Network 19
LD     SM0.0
MOVB   VB511, VB801
AENO
SRB    VB801, 2
AENO
MOVB   VB512, VB802
SLB    VB802, 4
Network 20
LDW<>  VW801, +0
AN     AS1:I9.4
=      MESS65:V408.0
Network 21
LD     AV取件完成:V512.6
O      AV放小件准备就绪:V511.0
ON     ST1_WORKING:M3.0
A      AS1:I9.4
=      MESS66:V408.1
Network 22
LD     SM0.0
MOVB   VB511, VB805
AENO
SRB    VB805, 5
AENO
MOVB   VB512, VB806
SLB    VB806, 4
Network 23
LDW<>  VW805, +0
AN     AS2:I9.5
=      MESS67:V408.2
Network 24
LD     SM0.0
MOVB   VB511, VB807
AENO
SLB    VB807, 4
AENO
MOVB   VB511, VB808
SRB    VB808, 5
Network 25
LDW<>  VW807, +0
ON     ST1_WORKING:M3.0
A      AS2:I9.5
=      MESS68:V408.3
Network 26
LD     SM0.0
MOVB   VB511, VB809
AENO
SRB    VB809, 2
AENO
MOVB   VB512, VB810
SLB    VB810, 4
Network 27
LDW<>  VW809, +0
AN     AS3:I10.6
=      MESS69:V408.4
Network 28
LD     AV取件完成:V512.6
O      AV放小件准备就绪:V511.0
ON     ST1_WORKING:M3.0
A      AS3:I10.6
=      MESS70:V408.5
Network 29
LD     SM0.0
MOVB   VB611, VB901
AENO
SRB    VB901, 2
AENO
MOVB   VB612, VB902
SLB    VB902, 4
Network 30
LDW<>  VW901, +0
AN     BS1:I3.4
=      MESS73:V409.0
Network 31
LD     BV取件完成:V612.6
O      BV放小件准备就绪:V611.0
ON     ST2_WORKING:M3.1
A      BS1:I3.4
=      MESS74:V409.1
Network 32
LD     SM0.0
MOVB   VB611, VB905
AENO
SRB    VB905, 5
AENO
MOVB   VB612, VB906
SLB    VB906, 4
Network 33
LDW<>  VW905, +0
AN     BS2:I3.5
=      MESS75:V409.2
Network 34
LD     SM0.0
MOVB   VB611, VB907
AENO
SLB    VB907, 4
AENO
MOVB   VB611, VB908
SRB    VB908, 5
Network 35
LDW<>  VW907, +0
ON     ST2_WORKING:M3.1
A      BS2:I3.5
=      MESS76:V409.3
Network 36
LD     SM0.0
MOVB   VB611, VB909
AENO
SRB    VB909, 2
AENO
MOVB   VB612, VB910
SLB    VB910, 4
Network 37
LDW<>  VW909, +0
AN     BS3:I4.6
=      MESS77:V409.4
Network 38
LD     BV取件完成:V612.6
O      BV放小件准备就绪:V611.0
ON     ST2_WORKING:M3.1
A      BS3:I4.6
=      MESS78:V409.5
Network 40
LD     A伺服就绪:I2.0
A      A_SRV_ON:Q11.0
AN     A_RSEEK_DONE:V545.1
=      MESS113:V414.0
Network 41
LDN    A伺服就绪:I2.0
=      MESS114:V414.1
Network 42
LD     A伺服就绪:I2.0
AN     A_SRV_ON:Q11.0
=      MESS115:V414.2
Network 43
LD     B_SRV_ON:Q11.2
A      B伺服就绪:I2.4
AN     B_RSEEK_DONE:V645.1
=      MESS116:V414.3
Network 44
LDN    B伺服就绪:I2.4
=      MESS117:V414.4
Network 45
LD     B伺服就绪:I2.4
AN     B_SRV_ON:Q11.2
=      MESS118:V414.5
Network 46
LD     BP_START:I0.6
EU
LDN    ST1_PASS:M2.4
AN     ST2_PASS:M2.6
A      INIT_FINISH:M2.2
LD     ST1_PASS:M2.4
AN     ST2_PASS:M2.6
A      INIT2_FINISH:M2.1
OLD
LDN    ST1_PASS:M2.4
A      ST2_PASS:M2.6
A      INIT1_FINISH:M2.0
OLD
ALD
A      R1_AUTO:I5.0
AN     R1_HOME:I5.4
S      MESS119:V414.6, 1
Network 47
LD     R1_HOME:I5.4
R      MESS119:V414.6, 1
Network 48
LD     BP_START:I0.6
EU
LDN    ST1_PASS:M2.4
AN     ST2_PASS:M2.6
A      INIT_FINISH:M2.2
LD     ST1_PASS:M2.4
AN     ST2_PASS:M2.6
A      INIT2_FINISH:M2.1
OLD
LDN    ST1_PASS:M2.4
A      ST2_PASS:M2.6
A      INIT1_FINISH:M2.0
OLD
ALD
A      R2_AUTO:I7.0
AN     R2_HOME:I7.4
=      MESS120:V414.7
Network 49
LD     R2_HOME:I7.4
R      MESS120:V414.7, 1
Network 50
LD     BP_AUTO:I0.5
AN     R1_AUTO:I5.0
=      MESS121:V415.0
Network 51
LD     BP_AUTO:I0.5
AN     R2_AUTO:I7.0
=      MESS122:V415.1
Network 52
LD     ATUOSTART:M10.2
A      R1_AUTO:I5.0
AN     R1_CYCLE_NO:I5.1
=      MESS123:V415.2
Network 53
LD     ATUOSTART:M10.2
A      R2_AUTO:I7.0
AN     R2_CYCLE_NO:I7.1
=      MESS124:V415.3
Network 54
LD     WORK_START:I0.1
EU
LDN    ST1_PASS:M2.4
AN     ST2_PASS:M2.6
A      INIT_FINISH:M2.2
LD     ST1_PASS:M2.4
AN     ST2_PASS:M2.6
A      INIT2_FINISH:M2.1
OLD
LDN    ST1_PASS:M2.4
A      ST2_PASS:M2.6
A      INIT1_FINISH:M2.0
OLD
ALD
A      BP_AUTO:I0.5
A      R1_AUTO:I5.0
AN     R2_工位1:I7.6
S      MESS125:V415.4, 1
Network 55
LD     HMI_AV1夹紧:V500.3
O      HMI_AV1放松:V501.3
O      HMI_AV2夹紧:V502.3
O      HMI_AV2放松:V503.3
O      HMI_AV3夹紧:V504.3
O      HMI_AV3放松:V505.3
EU
A      BP_MANUAL:I0.4
AN     R2_工位1:I7.6
S      MESS125:V415.4, 1
Network 56
LD     R2_工位1:I7.6
R      MESS125:V415.4, 1
Network 57
LD     WORK_START:I0.1
EU
LDN    ST1_PASS:M2.4
AN     ST2_PASS:M2.6
A      INIT_FINISH:M2.2
LD     ST1_PASS:M2.4
AN     ST2_PASS:M2.6
A      INIT2_FINISH:M2.1
OLD
LDN    ST1_PASS:M2.4
A      ST2_PASS:M2.6
A      INIT1_FINISH:M2.0
OLD
ALD
A      BP_AUTO:I0.5
A      R1_AUTO:I5.0
AN     R2_工位2:I7.7
S      MESS126:V415.5, 1
Network 58
LD     HMI_BV1夹紧:V600.3
O      HMI_BV1放松:V601.3
O      HMI_BV2夹紧:V602.3
O      HMI_BV2放松:V603.3
O      HMI_BV3夹紧:V604.3
O      HMI_BV3放松:V605.3
EU
A      BP_MANUAL:I0.4
AN     R2_工位2:I7.7
S      MESS126:V415.5, 1
Network 59
LD     R2_工位2:I7.7
R      MESS126:V415.5, 1
Network 60
LD     WORK_START:I0.1
EU
AN     ST1_PASS:M2.4
A      AV_HOME:M3.6
AN     AV未装件:V510.7
S      MESS127:V415.6, 1
Network 61
LD     AV未装件:V510.7
R      MESS127:V415.6, 1
Network 62
LD     WORK_START:I0.1
EU
AN     ST2_PASS:M2.6
A      BV_HOME:M3.7
AN     BV未装件:V610.7
S      MESS128:V415.7, 1
Network 63
LD     BV未装件:V610.7
R      MESS128:V415.7, 1
Network 64
LDN    R1_ES_OK:I5.5
=      MESS129:V416.0
Network 65
LDN    R2_ES_OK:I7.5
=      MESS130:V416.1
Network 66
LDN    ES_OK:I0.7
=      MESS131:V416.2
Network 67
LD     HMI_ES:I0.0
=      MESS132:V416.3
Network 68
LD     BP_ES:I1.0
=      MESS133:V416.4
Network 69
LDN    HMI_ES:I0.0
AN     BP_ES:I1.0
AN     ES_OK:I0.7
=      MESS134:V416.5
Network 70
LDN    AS_OK:I1.2
=      MESS135:V416.6
Network 71
LD     WORK_START:I0.1
EU
AN     ST1_WORKING:M3.0
AN     AV全部放松:V510.2
S      MESS137:V417.0, 1
Network 72
LD     AV全部放松:V510.2
R      MESS137:V417.0, 1
Network 73
LD     WORK_START:I0.1
EU
AN     ST2_WORKING:M3.1
AN     BV全部放松:V610.2
S      MESS138:V417.1, 1
Network 74
LD     BV全部放松:V610.2
R      MESS138:V417.1, 1
Network 75
LD     WORK_START:I0.1
EU
A      BV全部放松:V610.2
A      ST2_WORKING:M3.1
S      MESS139:V417.2, 1
Network 76
LDN    ST2_WORKING:M3.1
R      MESS139:V417.2, 1
Network 77
LD     HMI_RUN_FREE:M1.2
=      MESS145:V418.0
Network 78
LD     ST1_PASS:M2.4
=      MESS146:V418.1
Network 79
LD     ST2_PASS:M2.6
=      MESS147:V418.2
Network 80
LD     PAUSE:M2.3
=      MESS148:V418.3
Network 81
LD     FINISHED:M3.5
=      MESS149:V418.4
Network 85
LD     SM0.0
=      L60.0
LD     SM0.0
=      L63.7
LD     L60.0
CALL   SBR_25:SBR25, L63.7, +10
END_SUBROUTINE_BLOCK

SUBROUTINE_BLOCK chanpin:SBR41
TITLE=子程序注释
BEGIN
Network 2
//LD     HMI_产品选择2:V420.1
LDW<>  VW420, +0
A      A_SRV_ON:Q11.0
A      B_SRV_ON:Q11.2
A      A_RSEEK_DONE:V545.1
A      B_RSEEK_DONE:V645.1
MOVW   VW420, VW490
Network 3
//LD     HMI_产品选择3:V420.2
LD     放件确认:V465.0
MOVW   VW490, VW450
Network 4
LD     A_RSEEK_DONE:V545.1
EU
LD     B_RSEEK_DONE:V645.1
EU
OLD
MOVW   +0, VW450
Network 5
//LD     HMI_产品选择4:V420.3
LD     产品选择1:V450.0
AR=    A_RUN_C_POS:VD574, 833.6
A      A_RUN_DONE1:V541.3
=      A产品1:V460.0
Network 6
//LD     HMI_产品选择5:V420.4
LD     产品选择2:V450.1
AR=    A_RUN_C_POS:VD574, 833.6
A      A_RUN_DONE1:V541.3
=      A产品2:V460.1
Network 7
//LD     HMI_产品选择6:V420.5
LD     产品选择3:V450.2
AR=    A_RUN_C_POS:VD574, 784.0
A      A_RUN_DONE2:V541.6
=      A产品3:V460.2
Network 8
//LD     HMI_产品选择7:V420.6
LD     产品选择4:V450.3
AR=    A_RUN_C_POS:VD574, 784.0
A      A_RUN_DONE2:V541.6
=      A产品4:V460.3
Network 9
//LD     HMI_产品选择8:V420.7
LD     产品选择5:V450.4
AR=    A_RUN_C_POS:VD574, 734.5
A      A_RUN_DONE3:V542.1
=      A产品5:V460.4
Network 10
//LD     HMI_产品选择9:V421.0
LD     产品选择6:V450.5
AR=    A_RUN_C_POS:VD574, 734.5
A      A_RUN_DONE3:V542.1
=      A产品6:V460.5
Network 11
//LD     HMI_产品选择10:V421.1
LD     产品选择7:V450.6
AR=    A_RUN_C_POS:VD574, 385.0
A      A_RUN_DONE4:V542.4
=      A产品7:V460.6
Network 12
//LD     HMI_产品选择11:V421.2
LD     产品选择8:V450.7
AR=    A_RUN_C_POS:VD574, 385.0
A      A_RUN_DONE4:V542.4
=      A产品8:V460.7
Network 13
//LD     HMI_产品选择12:V421.3
LD     产品选择9:V451.0
AR=    A_RUN_C_POS:VD574, 827.0
A      A_RUN_DONE5:V542.7
=      A产品9:V461.0
Network 14
//LD     HMI_产品选择13:V421.4
LD     产品选择10:V451.1
AR=    A_RUN_C_POS:VD574, 827.0
A      A_RUN_DONE5:V542.7
=      A产品10:V461.1
Network 15
//LD     HMI_产品选择14:V421.5
LD     产品选择11:V451.2
AR=    A_RUN_C_POS:VD574, 780.8
A      A_RUN_DONE6:V543.2
=      A产品11:V461.2
Network 16
//LD     HMI_产品选择15:V421.6
LD     产品选择12:V451.3
AR=    A_RUN_C_POS:VD574, 731.5
A      A_RUN_DONE7:V543.5
=      A产品12:V461.3
Network 17
LD     产品选择13:V451.4
AR=    A_RUN_C_POS:VD574, 381.5
A      A_RUN_DONE8:V544.0
=      A产品13:V461.4
Network 18
LD     产品选择14:V451.5
AR=    A_RUN_C_POS:VD574, 381.5
A      A_RUN_DONE8:V544.0
=      A产品14:V461.5
Network 19
LD     产品选择15:V451.6
=      A产品15:V461.6
Network 20
// A1
Network 21
// A2
Network 22
// A3
Network 23
// A4
LD     产品选择1:V450.0
AR=    B_RUN_C_POS:VD674, 824.0
A      B_RUN_DONE1:V641.3
=      B产品1:V462.0
Network 24
// A5
LD     产品选择2:V450.1
AR=    B_RUN_C_POS:VD674, 824.0
A      B_RUN_DONE1:V641.3
=      B产品2:V462.1
Network 25
// A6
LD     产品选择3:V450.2
AR=    B_RUN_C_POS:VD674, 774.5
A      B_RUN_DONE2:V641.6
=      B产品3:V462.2
Network 26
// A7
LD     产品选择4:V450.3
AR=    B_RUN_C_POS:VD674, 774.5
A      B_RUN_DONE2:V641.6
=      B产品4:V462.3
Network 27
// A8
LD     产品选择5:V450.4
AR=    B_RUN_C_POS:VD674, 724.8
A      B_RUN_DONE3:V642.1
=      B产品5:V462.4
Network 28
// A9
LD     产品选择6:V450.5
AR=    B_RUN_C_POS:VD674, 724.8
A      B_RUN_DONE3:V642.1
=      B产品6:V462.5
Network 29
// A10
LD     产品选择7:V450.6
AR=    B_RUN_C_POS:VD674, 375.0
A      B_RUN_DONE4:V642.4
=      B产品7:V462.6
Network 30
// A11
LD     产品选择8:V450.7
AR=    B_RUN_C_POS:VD674, 375.0
A      B_RUN_DONE4:V642.4
=      B产品8:V462.7
Network 31
// A12
LD     产品选择9:V451.0
AR=    B_RUN_C_POS:VD674, 817.0
A      B_RUN_DONE5:V642.7
=      B产品9:V463.0
Network 32
// A13
LD     产品选择10:V451.1
AR=    B_RUN_C_POS:VD674, 817.0
A      B_RUN_DONE5:V642.7
=      B产品10:V463.1
Network 33
// A14
LD     产品选择11:V451.2
AR=    B_RUN_C_POS:VD674, 771.0
A      B_RUN_DONE6:V643.2
=      B产品11:V463.2
Network 34
// A15
LD     产品选择12:V451.3
AR=    B_RUN_C_POS:VD674, 721.5
A      B_RUN_DONE7:V643.5
=      B产品12:V463.3
Network 35
LD     产品选择13:V451.4
AR=    B_RUN_C_POS:VD674, 371.5
A      B_RUN_DONE8:V644.0
=      B产品13:V463.4
Network 36
LD     产品选择14:V451.5
AR=    B_RUN_C_POS:VD674, 371.5
A      B_RUN_DONE8:V644.0
=      B产品14:V463.5
Network 37
LD     产品选择15:V451.6
=      B产品15:V463.6
Network 38
// B1
Network 39
// B2
LD     A产品1:V460.0
A      B产品1:V462.0
R      产品组信号1:M12.0, 4
S      产品组信号1:M12.0, 1
Network 40
// B3
LD     A产品2:V460.1
A      B产品2:V462.1
R      产品组信号1:M12.0, 4
S      产品组信号2:M12.1, 1
Network 41
// B4
LD     A产品3:V460.2
A      B产品3:V462.2
R      产品组信号1:M12.0, 4
S      产品组信号1:M12.0, 2
Network 42
// B5
LD     A产品4:V460.3
A      B产品4:V462.3
R      产品组信号1:M12.0, 4
S      产品组信号3:M12.2, 1
Network 43
// B6
LD     A产品5:V460.4
A      B产品5:V462.4
R      产品组信号1:M12.0, 4
S      产品组信号1:M12.0, 1
S      产品组信号3:M12.2, 1
Network 44
// B7
LD     A产品6:V460.5
A      B产品6:V462.5
R      产品组信号1:M12.0, 4
S      产品组信号2:M12.1, 2
Network 45
// B8
LD     A产品7:V460.6
A      B产品7:V462.6
R      产品组信号1:M12.0, 4
S      产品组信号1:M12.0, 3
Network 46
// B9
LD     A产品8:V460.7
A      B产品8:V462.7
R      产品组信号1:M12.0, 4
S      产品组信号4:M12.3, 1
Network 47
// B10
LD     A产品9:V461.0
A      B产品9:V463.0
R      产品组信号1:M12.0, 4
S      产品组信号1:M12.0, 1
S      产品组信号4:M12.3, 1
Network 48
// B11
LD     A产品10:V461.1
A      B产品10:V463.1
R      产品组信号1:M12.0, 4
S      产品组信号2:M12.1, 1
S      产品组信号4:M12.3, 1
Network 49
// B12
LD     A产品11:V461.2
A      B产品11:V463.2
R      产品组信号1:M12.0, 4
S      产品组信号1:M12.0, 2
S      产品组信号4:M12.3, 1
Network 50
// B13
LD     A产品12:V461.3
A      B产品12:V463.3
R      产品组信号1:M12.0, 4
S      产品组信号3:M12.2, 2
Network 51
// B14
LD     A产品13:V461.4
A      B产品13:V463.4
R      产品组信号1:M12.0, 4
S      产品组信号1:M12.0, 1
S      产品组信号3:M12.2, 2
Network 52
// B15
LD     A产品14:V461.5
A      B产品14:V463.5
R      产品组信号1:M12.0, 4
S      产品组信号2:M12.1, 3
Network 53
LD     A产品15:V461.6
A      B产品15:V463.6
S      产品组信号1:M12.0, 4
Network 55
LD     SM0.0
MOVB   QB7, 产品提示:VB470
AENO
SLB    产品提示:VB470, 2
AENO
MOVB   产品提示:VB470, 产品选择显示:VB480
SRB    产品选择显示:VB480, 4
END_SUBROUTINE_BLOCK

// (further data pages could not be read)
